(* PLC project Export.project, CODESYS CODESYS V3.5 SP19 Patch 7 *)
(* stored: creationDateTime 2025-04-03T07:54:30.183, modificationDateTime 2025-04-03T07:54:30.183 *)

VAR_GLOBAL  (* GVL_ClimateControl *)
  typClimateControllerInterfaceRoom401 : typMultiModeClimateControl_00_01;
  typClimateControllerInterfaceRoom406 : typMultiModeClimateControl_00_01;
  typClimateControllerInterfaceRoom407 : typMultiModeClimateControl_00_01;
  typClimateControllerInterfaceRoom408 : typMultiModeClimateControl_00_01;
  typClimateControllerInterfaceRoom409 : typMultiModeClimateControl_00_01;
  typClimateControllerInterfaceRoom464 : typMultiModeClimateControl_00_01;
  typClimateControllerInterfaceRoom415 : typMultiModeClimateControl_00_01;
  typClimateControllerInterfaceRoom422 : typMultiModeClimateControl_00_01;
  typClimateControllerInterfaceRoom426_1 : typMultiModeClimateControl_00_01;
  typClimateControllerInterfaceRoom426_2 : typMultiModeClimateControl_00_01;
  typClimateControllerInterfaceRoom426_3 : typMultiModeClimateControl_00_01;
  typClimateControllerInterfaceRoom528 : typMultiModeClimateControl_00_01;
  typClimateControllerInterfaceRoom523 : typMultiModeClimateControl_00_01;
  typClimateControllerInterfaceRoom531 : typMultiModeClimateControl_00_01;
  typClimateControllerInterfaceRoom535_1 : typMultiModeClimateControl_00_01;
  typClimateControllerInterfaceRoom535_2 : typMultiModeClimateControl_00_01;
  typClimateControllerInterfaceRoom535_3 : typMultiModeClimateControl_00_01;
  typClimateControllerInterfaceRoom536 : typMultiModeClimateControl_00_01;
  typClimateControllerInterfaceRoom543 : typMultiModeClimateControl_00_01;
  typClimateControllerInterfaceRoom547_1 : typMultiModeClimateControl_00_01;
  typClimateControllerInterfaceRoom547_2 : typMultiModeClimateControl_00_01;
  typClimateControllerInterfaceRoom544 : typMultiModeClimateControl_00_01;
  SLETT_MEG : BOOL;  (* Kopier til PersistentVars! *)
  typClimateControllerSettingsRoom401 : typMultiModeClimateControlSettings_00_01;
  typClimateControllerSettingsRoom406 : typMultiModeClimateControlSettings_00_01;
  typClimateControllerSettingsRoom407 : typMultiModeClimateControlSettings_00_01;
  typClimateControllerSettingsRoom408 : typMultiModeClimateControlSettings_00_01;
  typClimateControllerSettingsRoom409 : typMultiModeClimateControlSettings_00_01;
  typClimateControllerSettingsRoom464 : typMultiModeClimateControlSettings_00_01;
  typClimateControllerSettingsRoom415 : typMultiModeClimateControlSettings_00_01;
  typClimateControllerSettingsRoom422 : typMultiModeClimateControlSettings_00_01;
  typClimateControllerSettingsRoom426_1 : typMultiModeClimateControlSettings_00_01;
  typClimateControllerSettingsRoom426_2 : typMultiModeClimateControlSettings_00_01;
  typClimateControllerSettingsRoom426_3 : typMultiModeClimateControlSettings_00_01;
  typClimateControllerSettingsRoom528 : typMultiModeClimateControlSettings_00_01;
  typClimateControllerSettingsRoom523 : typMultiModeClimateControlSettings_00_01;
  typClimateControllerSettingsRoom531 : typMultiModeClimateControlSettings_00_01;
  typClimateControllerSettingsRoom535_1 : typMultiModeClimateControlSettings_00_01;
  typClimateControllerSettingsRoom535_2 : typMultiModeClimateControlSettings_00_01;
  typClimateControllerSettingsRoom535_3 : typMultiModeClimateControlSettings_00_01;
  typClimateControllerSettingsRoom536 : typMultiModeClimateControlSettings_00_01;
  typClimateControllerSettingsRoom543 : typMultiModeClimateControlSettings_00_01;
  typClimateControllerSettingsRoom547_1 : typMultiModeClimateControlSettings_00_01;
  typClimateControllerSettingsRoom547_2 : typMultiModeClimateControlSettings_00_01;
  typClimateControllerSettingsRoom544 : typMultiModeClimateControlSettings_00_01;
END_VAR

VAR_GLOBAL  (* GVL_BACnet *)
  C_5640_501_06_RBA01_D_R0401 : FbBinaryOutput_Medium (0) := (                _sDescription := 'Tilstedeværelsesdetektor',                 _sActiveText := 'Tilstedeværelse',                 _sInactiveText := 'Ingen tilstedeværelse'           );
  C_5640_501_06_RTC01_MV_R0401 : FbAnalogInput_Large (0) := (                _sDescription := 'Målt temperatur',                 _rCov_Increment := 0.1,                 _eUnits := WagoTypesBacnet.eBACnetUnits.UNIT_DEGREES_C,                 _rHighLimit := 28,                 _ILimitEnable := ( xLowLimitReporting := FALSE, xHighLimitReporting := TRUE ),                 _udiNotificationClass := 22           );
  C_5640_501_06_RTC01_SPV_R0401 : FbAnalogValue_Medium (0) := (                _sDescription := 'Arbeidende settpunkt',                 _rCov_Increment := 0.1,                 _eUnits := WagoTypesBacnet.eBACnetUnits.UNIT_DEGREES_C           );
  C_5640_501_06_RTC01_SPV_Komf_R0401 : FbAnalogValue_Medium (1) := (                _sDescription := 'Settpunkt komfort',                 _rCov_Increment := 0.1,                 _eUnits := WagoTypesBacnet.eBACnetUnits.UNIT_DEGREES_C           );
  C_5640_501_06_RTC01_SPV_Stdb_R0401 : FbAnalogValue_Medium (2) := (                _sDescription := 'Settpunkt Standby',                 _rCov_Increment := 0.1,                 _eUnits := WagoTypesBacnet.eBACnetUnits.UNIT_DEGREES_C           );
  C_5640_501_06_RTC01_SPV_Natt_R0401 : FbAnalogValue_Medium (3) := (                _sDescription := 'Settpunkt Natt',                 _rCov_Increment := 0.1,                 _eUnits := WagoTypesBacnet.eBACnetUnits.UNIT_DEGREES_C           );
  C_5640_501_06_RTC01_MOD_FB_R0401 : FbMultiStateValue_Large (0) := (                _sDescription := 'Tilbakemelding driftmodus',                 _udiNumberOfStates := 5,                 _xEventDetectionEnable := FALSE,                 _udiNotificationClass := 99           );
  C_5640_501_06_RTC01_KMD_MSV_R0401 : FbMultiStateValue_Large (1) := (                _sDescription := 'Kalender',                 _udiNumberOfStates := 10,                 _xEventDetectionEnable := FALSE,                 _udiNotificationClass := 99           );
  C_5640_501_06_RTC01_SP_Tid_Stdb_R0401 : FbAnalogValue_Medium (4) := (                _sDescription := 'Utløpstid tilstedeværelse',                 _rCov_Increment := 1,                 _eUnits := WagoTypesBacnet.eBACnetUnits.UNIT_MINUTES           );
  C_5640_501_06_RYA601_SP_R0401 : FbAnalogValue_Medium (5) := (                _sDescription := 'Settpunkt',                 _rCov_Increment := 1,                 _eUnits := WagoTypesBacnet.eBACnetUnits.UNIT_PARTS_PER_MILLION           );
  C_5640_501_06_RYA601_MV_R0401 : FbAnalogInput_Large (1) := (                _sDescription := 'Målt CO2-konsentrasjon',                 _rCov_Increment := 1,                 _eUnits := WagoTypesBacnet.eBACnetUnits.UNIT_PARTS_PER_MILLION,                 _rHighLimit := 1000,                 _ILimitEnable := ( xLowLimitReporting := FALSE, xHighLimitReporting := TRUE ),                 _udiNotificationClass := 22           );
  C_5640_501_06_SBB01_C_R0401 : FbAnalogOutput_Medium (0) := (                _sDescription := 'Pådrag varmeorgan',                 _rCov_Increment := 1,                 _eUnits := WagoTypesBacnet.eBACnetUnits.UNIT_PERCENT           );
  C_5640_501_06_RBA01_D_R0406 : FbBinaryOutput_Medium (1) := (                _sDescription := 'Tilstedeværelsesdetektor',                 _sActiveText := 'Tilstedeværelse',                 _sInactiveText := 'Ingen tilstedeværelse'           );
  C_5640_501_06_RTC01_MV_R0406 : FbAnalogInput_Large (2) := (                _sDescription := 'Målt temperatur',                 _rCov_Increment := 0.1,                 _eUnits := WagoTypesBacnet.eBACnetUnits.UNIT_DEGREES_C,                 _rHighLimit := 28,                 _ILimitEnable := ( xLowLimitReporting := FALSE, xHighLimitReporting := TRUE ),                 _udiNotificationClass := 22           );
  C_5640_501_06_RTC01_SPV_R0406 : FbAnalogValue_Medium (6) := (                _sDescription := 'Arbeidende settpunkt',                 _rCov_Increment := 0.1,                 _eUnits := WagoTypesBacnet.eBACnetUnits.UNIT_DEGREES_C           );
  C_5640_501_06_RTC01_SPV_Komf_R0406 : FbAnalogValue_Medium (7) := (                _sDescription := 'Settpunkt komfort',                 _rCov_Increment := 0.1,                 _eUnits := WagoTypesBacnet.eBACnetUnits.UNIT_DEGREES_C           );
  C_5640_501_06_RTC01_SPV_Stdb_R0406 : FbAnalogValue_Medium (8) := (                _sDescription := 'Settpunkt Standby',                 _rCov_Increment := 0.1,                 _eUnits := WagoTypesBacnet.eBACnetUnits.UNIT_DEGREES_C           );
  C_5640_501_06_RTC01_SPV_Natt_R0406 : FbAnalogValue_Medium (9) := (                _sDescription := 'Settpunkt Natt',                 _rCov_Increment := 0.1,                 _eUnits := WagoTypesBacnet.eBACnetUnits.UNIT_DEGREES_C           );
  C_5640_501_06_RTC01_MOD_FB_R0406 : FbMultiStateValue_Large (2) := (                _sDescription := 'Tilbakemelding driftmodus',                 _udiNumberOfStates := 5,                 _xEventDetectionEnable := FALSE,                 _udiNotificationClass := 99           );
  C_5640_501_06_RTC01_KMD_MSV_R0406 : FbMultiStateValue_Large (3) := (                _sDescription := 'Kalender',                 _udiNumberOfStates := 10,                 _xEventDetectionEnable := FALSE,                 _udiNotificationClass := 99           );
  C_5640_501_06_RTC01_SP_Tid_Stdb_R0406 : FbAnalogValue_Medium (10) := (                _sDescription := 'Utløpstid tilstedeværelse',                 _rCov_Increment := 1,                 _eUnits := WagoTypesBacnet.eBACnetUnits.UNIT_MINUTES           );
  C_5640_501_06_RYA601_SP_R0406 : FbAnalogValue_Medium (11) := (                _sDescription := 'Settpunkt',                 _rCov_Increment := 1,                 _eUnits := WagoTypesBacnet.eBACnetUnits.UNIT_PARTS_PER_MILLION           );
  C_5640_501_06_RYA601_MV_R0406 : FbAnalogInput_Large (3) := (                _sDescription := 'Målt CO2-konsentrasjon',                 _rCov_Increment := 1,                 _eUnits := WagoTypesBacnet.eBACnetUnits.UNIT_PARTS_PER_MILLION,                 _rHighLimit := 1000,                 _ILimitEnable := ( xLowLimitReporting := FALSE, xHighLimitReporting := TRUE ),                 _udiNotificationClass := 22           );
  C_5640_501_06_SBB01_C_R0406 : FbAnalogOutput_Medium (1) := (                _sDescription := 'Pådrag varmeorgan',                 _rCov_Increment := 1,                 _eUnits := WagoTypesBacnet.eBACnetUnits.UNIT_PERCENT           );
  C_5640_501_06_RBA01_D_R0407 : FbBinaryOutput_Medium (2) := (                _sDescription := 'Tilstedeværelsesdetektor',                 _sActiveText := 'Tilstedeværelse',                 _sInactiveText := 'Ingen tilstedeværelse'           );
  C_5640_501_06_RTC01_MV_R0407 : FbAnalogInput_Large (4) := (                _sDescription := 'Målt temperatur',                 _rCov_Increment := 0.1,                 _eUnits := WagoTypesBacnet.eBACnetUnits.UNIT_DEGREES_C,                 _rHighLimit := 28,                 _ILimitEnable := ( xLowLimitReporting := FALSE, xHighLimitReporting := TRUE ),                 _udiNotificationClass := 22           );
  C_5640_501_06_RTC01_SPV_R0407 : FbAnalogValue_Medium (12) := (                _sDescription := 'Arbeidende settpunkt',                 _rCov_Increment := 0.1,                 _eUnits := WagoTypesBacnet.eBACnetUnits.UNIT_DEGREES_C           );
  C_5640_501_06_RTC01_SPV_Komf_R0407 : FbAnalogValue_Medium (13) := (                _sDescription := 'Settpunkt komfort',                 _rCov_Increment := 0.1,                 _eUnits := WagoTypesBacnet.eBACnetUnits.UNIT_DEGREES_C           );
  C_5640_501_06_RTC01_SPV_Stdb_R0407 : FbAnalogValue_Medium (14) := (                _sDescription := 'Settpunkt Standby',                 _rCov_Increment := 0.1,                 _eUnits := WagoTypesBacnet.eBACnetUnits.UNIT_DEGREES_C           );
  C_5640_501_06_RTC01_SPV_Natt_R0407 : FbAnalogValue_Medium (15) := (                _sDescription := 'Settpunkt Natt',                 _rCov_Increment := 0.1,                 _eUnits := WagoTypesBacnet.eBACnetUnits.UNIT_DEGREES_C           );
  C_5640_501_06_RTC01_MOD_FB_R0407 : FbMultiStateValue_Large (4) := (                _sDescription := 'Tilbakemelding driftmodus',                 _udiNumberOfStates := 5,                 _xEventDetectionEnable := FALSE,                 _udiNotificationClass := 99           );
  C_5640_501_06_RTC01_KMD_MSV_R0407 : FbMultiStateValue_Large (5) := (                _sDescription := 'Kalender',                 _udiNumberOfStates := 10,                 _xEventDetectionEnable := FALSE,                 _udiNotificationClass := 99           );
  C_5640_501_06_RTC01_SP_Tid_Stdb_R0407 : FbAnalogValue_Medium (16) := (                _sDescription := 'Utløpstid tilstedeværelse',                 _rCov_Increment := 1,                 _eUnits := WagoTypesBacnet.eBACnetUnits.UNIT_MINUTES           );
  C_5640_501_06_RYA601_SP_R0407 : FbAnalogValue_Medium (17) := (                _sDescription := 'Settpunkt',                 _rCov_Increment := 1,                 _eUnits := WagoTypesBacnet.eBACnetUnits.UNIT_PARTS_PER_MILLION           );
  C_5640_501_06_RYA601_MV_R0407 : FbAnalogInput_Large (5) := (                _sDescription := 'Målt CO2-konsentrasjon',                 _rCov_Increment := 1,                 _eUnits := WagoTypesBacnet.eBACnetUnits.UNIT_PARTS_PER_MILLION,                 _rHighLimit := 1000,                 _ILimitEnable := ( xLowLimitReporting := FALSE, xHighLimitReporting := TRUE ),                 _udiNotificationClass := 22           );
  C_5640_501_06_SBB01_C_R0407 : FbAnalogOutput_Medium (2) := (                _sDescription := 'Pådrag varmeorgan',                 _rCov_Increment := 1,                 _eUnits := WagoTypesBacnet.eBACnetUnits.UNIT_PERCENT           );
  C_5640_501_06_RBA01_D_R0408 : FbBinaryOutput_Medium (3) := (                _sDescription := 'Tilstedeværelsesdetektor',                 _sActiveText := 'Tilstedeværelse',                 _sInactiveText := 'Ingen tilstedeværelse'           );
  C_5640_501_06_RTC01_MV_R0408 : FbAnalogInput_Large (6) := (                _sDescription := 'Målt temperatur',                 _rCov_Increment := 0.1,                 _eUnits := WagoTypesBacnet.eBACnetUnits.UNIT_DEGREES_C,                 _rHighLimit := 28,                 _ILimitEnable := ( xLowLimitReporting := FALSE, xHighLimitReporting := TRUE ),                 _udiNotificationClass := 22           );
  C_5640_501_06_RTC01_SPV_R0408 : FbAnalogValue_Medium (18) := (                _sDescription := 'Arbeidende settpunkt',                 _rCov_Increment := 0.1,                 _eUnits := WagoTypesBacnet.eBACnetUnits.UNIT_DEGREES_C           );
  C_5640_501_06_RTC01_SPV_Komf_R0408 : FbAnalogValue_Medium (19) := (                _sDescription := 'Settpunkt komfort',                 _rCov_Increment := 0.1,                 _eUnits := WagoTypesBacnet.eBACnetUnits.UNIT_DEGREES_C           );
  C_5640_501_06_RTC01_SPV_Stdb_R0408 : FbAnalogValue_Medium (20) := (                _sDescription := 'Settpunkt Standby',                 _rCov_Increment := 0.1,                 _eUnits := WagoTypesBacnet.eBACnetUnits.UNIT_DEGREES_C           );
  C_5640_501_06_RTC01_SPV_Natt_R0408 : FbAnalogValue_Medium (21) := (                _sDescription := 'Settpunkt Natt',                 _rCov_Increment := 0.1,                 _eUnits := WagoTypesBacnet.eBACnetUnits.UNIT_DEGREES_C           );
  C_5640_501_06_RTC01_MOD_FB_R0408 : FbMultiStateValue_Large (6) := (                _sDescription := 'Tilbakemelding driftmodus',                 _udiNumberOfStates := 5,                 _xEventDetectionEnable := FALSE,                 _udiNotificationClass := 99           );
  C_5640_501_06_RTC01_KMD_MSV_R0408 : FbMultiStateValue_Large (7) := (                _sDescription := 'Kalender',                 _udiNumberOfStates := 10,                 _xEventDetectionEnable := FALSE,                 _udiNotificationClass := 99           );
  C_5640_501_06_RTC01_SP_Tid_Stdb_R0408 : FbAnalogValue_Medium (22) := (                _sDescription := 'Utløpstid tilstedeværelse',                 _rCov_Increment := 1,                 _eUnits := WagoTypesBacnet.eBACnetUnits.UNIT_MINUTES           );
  C_5640_501_06_RYA601_SP_R0408 : FbAnalogValue_Medium (23) := (                _sDescription := 'Settpunkt',                 _rCov_Increment := 1,                 _eUnits := WagoTypesBacnet.eBACnetUnits.UNIT_PARTS_PER_MILLION           );
  C_5640_501_06_RYA601_MV_R0408 : FbAnalogInput_Large (7) := (                _sDescription := 'Målt CO2-konsentrasjon',                 _rCov_Increment := 1,                 _eUnits := WagoTypesBacnet.eBACnetUnits.UNIT_PARTS_PER_MILLION,                 _rHighLimit := 1000,                 _ILimitEnable := ( xLowLimitReporting := FALSE, xHighLimitReporting := TRUE ),                 _udiNotificationClass := 22           );
  C_5640_501_06_SBB01_C_R0408 : FbAnalogOutput_Medium (3) := (                _sDescription := 'Pådrag varmeorgan',                 _rCov_Increment := 1,                 _eUnits := WagoTypesBacnet.eBACnetUnits.UNIT_PERCENT           );
  C_5640_501_06_RBA01_D_R0409 : FbBinaryOutput_Medium (4) := (                _sDescription := 'Tilstedeværelsesdetektor',                 _sActiveText := 'Tilstedeværelse',                 _sInactiveText := 'Ingen tilstedeværelse'           );
  C_5640_501_06_RTC01_MV_R0409 : FbAnalogInput_Large (8) := (                _sDescription := 'Målt temperatur',                 _rCov_Increment := 0.1,                 _eUnits := WagoTypesBacnet.eBACnetUnits.UNIT_DEGREES_C,                 _rHighLimit := 28,                 _ILimitEnable := ( xLowLimitReporting := FALSE, xHighLimitReporting := TRUE ),                 _udiNotificationClass := 22           );
  C_5640_501_06_RTC01_SPV_R0409 : FbAnalogValue_Medium (24) := (                _sDescription := 'Arbeidende settpunkt',                 _rCov_Increment := 0.1,                 _eUnits := WagoTypesBacnet.eBACnetUnits.UNIT_DEGREES_C           );
  C_5640_501_06_RTC01_SPV_Komf_R0409 : FbAnalogValue_Medium (25) := (                _sDescription := 'Settpunkt komfort',                 _rCov_Increment := 0.1,                 _eUnits := WagoTypesBacnet.eBACnetUnits.UNIT_DEGREES_C           );
  C_5640_501_06_RTC01_SPV_Stdb_R0409 : FbAnalogValue_Medium (26) := (                _sDescription := 'Settpunkt Standby',                 _rCov_Increment := 0.1,                 _eUnits := WagoTypesBacnet.eBACnetUnits.UNIT_DEGREES_C           );
  C_5640_501_06_RTC01_SPV_Natt_R0409 : FbAnalogValue_Medium (27) := (                _sDescription := 'Settpunkt Natt',                 _rCov_Increment := 0.1,                 _eUnits := WagoTypesBacnet.eBACnetUnits.UNIT_DEGREES_C           );
  C_5640_501_06_RTC01_MOD_FB_R0409 : FbMultiStateValue_Large (8) := (                _sDescription := 'Tilbakemelding driftmodus',                 _udiNumberOfStates := 5,                 _xEventDetectionEnable := FALSE,                 _udiNotificationClass := 99           );
  C_5640_501_06_RTC01_KMD_MSV_R0409 : FbMultiStateValue_Large (9) := (                _sDescription := 'Kalender',                 _udiNumberOfStates := 10,                 _xEventDetectionEnable := FALSE,                 _udiNotificationClass := 99           );
  C_5640_501_06_RTC01_SP_Tid_Stdb_R0409 : FbAnalogValue_Medium (28) := (                _sDescription := 'Utløpstid tilstedeværelse',                 _rCov_Increment := 1,                 _eUnits := WagoTypesBacnet.eBACnetUnits.UNIT_MINUTES           );
  C_5640_501_06_RYA601_SP_R0409 : FbAnalogValue_Medium (29) := (                _sDescription := 'Settpunkt',                 _rCov_Increment := 1,                 _eUnits := WagoTypesBacnet.eBACnetUnits.UNIT_PARTS_PER_MILLION           );
  C_5640_501_06_RYA601_MV_R0409 : FbAnalogInput_Large (9) := (                _sDescription := 'Målt CO2-konsentrasjon',                 _rCov_Increment := 1,                 _eUnits := WagoTypesBacnet.eBACnetUnits.UNIT_PARTS_PER_MILLION,                 _rHighLimit := 1000,                 _ILimitEnable := ( xLowLimitReporting := FALSE, xHighLimitReporting := TRUE ),                 _udiNotificationClass := 22           );
  C_5640_501_06_SBB01_C_R0409 : FbAnalogOutput_Medium (4) := (                _sDescription := 'Pådrag varmeorgan',                 _rCov_Increment := 1,                 _eUnits := WagoTypesBacnet.eBACnetUnits.UNIT_PERCENT           );
  C_5640_501_06_RBA01_D_R0464 : FbBinaryOutput_Medium (5) := (                _sDescription := 'Tilstedeværelsesdetektor',                 _sActiveText := 'Tilstedeværelse',                 _sInactiveText := 'Ingen tilstedeværelse'           );
  C_5640_501_06_RTC01_MV_R0464 : FbAnalogInput_Large (10) := (                _sDescription := 'Målt temperatur',                 _rCov_Increment := 0.1,                 _eUnits := WagoTypesBacnet.eBACnetUnits.UNIT_DEGREES_C,                 _rHighLimit := 28,                 _ILimitEnable := ( xLowLimitReporting := FALSE, xHighLimitReporting := TRUE ),                 _udiNotificationClass := 22           );
  C_5640_501_06_RTC01_SPV_R0464 : FbAnalogValue_Medium (30) := (                _sDescription := 'Arbeidende settpunkt',                 _rCov_Increment := 0.1,                 _eUnits := WagoTypesBacnet.eBACnetUnits.UNIT_DEGREES_C           );
  C_5640_501_06_RTC01_SPV_Komf_R0464 : FbAnalogValue_Medium (31) := (                _sDescription := 'Settpunkt komfort',                 _rCov_Increment := 0.1,                 _eUnits := WagoTypesBacnet.eBACnetUnits.UNIT_DEGREES_C           );
  C_5640_501_06_RTC01_SPV_Stdb_R0464 : FbAnalogValue_Medium (32) := (                _sDescription := 'Settpunkt Standby',                 _rCov_Increment := 0.1,                 _eUnits := WagoTypesBacnet.eBACnetUnits.UNIT_DEGREES_C           );
  C_5640_501_06_RTC01_SPV_Natt_R0464 : FbAnalogValue_Medium (33) := (                _sDescription := 'Settpunkt Natt',                 _rCov_Increment := 0.1,                 _eUnits := WagoTypesBacnet.eBACnetUnits.UNIT_DEGREES_C           );
  C_5640_501_06_RTC01_MOD_FB_R0464 : FbMultiStateValue_Large (10) := (                _sDescription := 'Tilbakemelding driftmodus',                 _udiNumberOfStates := 5,                 _xEventDetectionEnable := FALSE,                 _udiNotificationClass := 99           );
  C_5640_501_06_RTC01_KMD_MSV_R0464 : FbMultiStateValue_Large (11) := (                _sDescription := 'Kalender',                 _udiNumberOfStates := 10,                 _xEventDetectionEnable := FALSE,                 _udiNotificationClass := 99           );
  C_5640_501_06_RTC01_SP_Tid_Stdb_R0464 : FbAnalogValue_Medium (34) := (                _sDescription := 'Utløpstid tilstedeværelse',                 _rCov_Increment := 1,                 _eUnits := WagoTypesBacnet.eBACnetUnits.UNIT_MINUTES           );
  C_5640_501_06_RYA601_SP_R0464 : FbAnalogValue_Medium (35) := (                _sDescription := 'Settpunkt',                 _rCov_Increment := 1,                 _eUnits := WagoTypesBacnet.eBACnetUnits.UNIT_PARTS_PER_MILLION           );
  C_5640_501_06_RYA601_MV_R0464 : FbAnalogInput_Large (11) := (                _sDescription := 'Målt CO2-konsentrasjon',                 _rCov_Increment := 1,                 _eUnits := WagoTypesBacnet.eBACnetUnits.UNIT_PARTS_PER_MILLION,                 _rHighLimit := 1000,                 _ILimitEnable := ( xLowLimitReporting := FALSE, xHighLimitReporting := TRUE ),                 _udiNotificationClass := 22           );
  C_5640_501_06_SBB01_C_R0464 : FbAnalogOutput_Medium (5) := (                _sDescription := 'Pådrag varmeorgan',                 _rCov_Increment := 1,                 _eUnits := WagoTypesBacnet.eBACnetUnits.UNIT_PERCENT           );
  C_5640_501_06_RBA01_D_R0415 : FbBinaryOutput_Medium (6) := (                _sDescription := 'Tilstedeværelsesdetektor',                 _sActiveText := 'Tilstedeværelse',                 _sInactiveText := 'Ingen tilstedeværelse'           );
  C_5640_501_06_RTC01_MV_R0415 : FbAnalogInput_Large (12) := (                _sDescription := 'Målt temperatur',                 _rCov_Increment := 0.1,                 _eUnits := WagoTypesBacnet.eBACnetUnits.UNIT_DEGREES_C,                 _rHighLimit := 28,                 _ILimitEnable := ( xLowLimitReporting := FALSE, xHighLimitReporting := TRUE ),                 _udiNotificationClass := 22           );
  C_5640_501_06_RTC01_SPV_R0415 : FbAnalogValue_Medium (36) := (                _sDescription := 'Arbeidende settpunkt',                 _rCov_Increment := 0.1,                 _eUnits := WagoTypesBacnet.eBACnetUnits.UNIT_DEGREES_C           );
  C_5640_501_06_RTC01_SPV_Komf_R0415 : FbAnalogValue_Medium (37) := (                _sDescription := 'Settpunkt komfort',                 _rCov_Increment := 0.1,                 _eUnits := WagoTypesBacnet.eBACnetUnits.UNIT_DEGREES_C           );
  C_5640_501_06_RTC01_SPV_Stdb_R0415 : FbAnalogValue_Medium (38) := (                _sDescription := 'Settpunkt Standby',                 _rCov_Increment := 0.1,                 _eUnits := WagoTypesBacnet.eBACnetUnits.UNIT_DEGREES_C           );
  C_5640_501_06_RTC01_SPV_Natt_R0415 : FbAnalogValue_Medium (39) := (                _sDescription := 'Settpunkt Natt',                 _rCov_Increment := 0.1,                 _eUnits := WagoTypesBacnet.eBACnetUnits.UNIT_DEGREES_C           );
  C_5640_501_06_RTC01_MOD_FB_R0415 : FbMultiStateValue_Large (12) := (                _sDescription := 'Tilbakemelding driftmodus',                 _udiNumberOfStates := 5,                 _xEventDetectionEnable := FALSE,                 _udiNotificationClass := 99           );
  C_5640_501_06_RTC01_KMD_MSV_R0415 : FbMultiStateValue_Large (13) := (                _sDescription := 'Kalender',                 _udiNumberOfStates := 10,                 _xEventDetectionEnable := FALSE,                 _udiNotificationClass := 99           );
  C_5640_501_06_RTC01_SP_Tid_Stdb_R0415 : FbAnalogValue_Medium (40) := (                _sDescription := 'Utløpstid tilstedeværelse',                 _rCov_Increment := 1,                 _eUnits := WagoTypesBacnet.eBACnetUnits.UNIT_MINUTES           );
  C_5640_501_06_RYA601_SP_R0415 : FbAnalogValue_Medium (41) := (                _sDescription := 'Settpunkt',                 _rCov_Increment := 1,                 _eUnits := WagoTypesBacnet.eBACnetUnits.UNIT_PARTS_PER_MILLION           );
  C_5640_501_06_RYA601_MV_R0415 : FbAnalogInput_Large (13) := (                _sDescription := 'Målt CO2-konsentrasjon',                 _rCov_Increment := 1,                 _eUnits := WagoTypesBacnet.eBACnetUnits.UNIT_PARTS_PER_MILLION,                 _rHighLimit := 1000,                 _ILimitEnable := ( xLowLimitReporting := FALSE, xHighLimitReporting := TRUE ),                 _udiNotificationClass := 22           );
  C_5640_501_06_SBB01_C_R0415 : FbAnalogOutput_Medium (6) := (                _sDescription := 'Pådrag varmeorgan',                 _rCov_Increment := 1,                 _eUnits := WagoTypesBacnet.eBACnetUnits.UNIT_PERCENT           );
  C_5640_501_06_RBA01_D_R0422 : FbBinaryOutput_Medium (7) := (                _sDescription := 'Tilstedeværelsesdetektor',                 _sActiveText := 'Tilstedeværelse',                 _sInactiveText := 'Ingen tilstedeværelse'           );
  C_5640_501_06_RTC01_MV_R0422 : FbAnalogInput_Large (14) := (                _sDescription := 'Målt temperatur',                 _rCov_Increment := 0.1,                 _eUnits := WagoTypesBacnet.eBACnetUnits.UNIT_DEGREES_C,                 _rHighLimit := 28,                 _ILimitEnable := ( xLowLimitReporting := FALSE, xHighLimitReporting := TRUE ),                 _udiNotificationClass := 22           );
  C_5640_501_06_RTC01_SPV_R0422 : FbAnalogValue_Medium (42) := (                _sDescription := 'Arbeidende settpunkt',                 _rCov_Increment := 0.1,                 _eUnits := WagoTypesBacnet.eBACnetUnits.UNIT_DEGREES_C           );
  C_5640_501_06_RTC01_SPV_Komf_R0422 : FbAnalogValue_Medium (43) := (                _sDescription := 'Settpunkt komfort',                 _rCov_Increment := 0.1,                 _eUnits := WagoTypesBacnet.eBACnetUnits.UNIT_DEGREES_C           );
  C_5640_501_06_RTC01_SPV_Stdb_R0422 : FbAnalogValue_Medium (44) := (                _sDescription := 'Settpunkt Standby',                 _rCov_Increment := 0.1,                 _eUnits := WagoTypesBacnet.eBACnetUnits.UNIT_DEGREES_C           );
  C_5640_501_06_RTC01_SPV_Natt_R0422 : FbAnalogValue_Medium (45) := (                _sDescription := 'Settpunkt Natt',                 _rCov_Increment := 0.1,                 _eUnits := WagoTypesBacnet.eBACnetUnits.UNIT_DEGREES_C           );
  C_5640_501_06_RTC01_MOD_FB_R0422 : FbMultiStateValue_Large (14) := (                _sDescription := 'Tilbakemelding driftmodus',                 _udiNumberOfStates := 5,                 _xEventDetectionEnable := FALSE,                 _udiNotificationClass := 99           );
  C_5640_501_06_RTC01_KMD_MSV_R0422 : FbMultiStateValue_Large (15) := (                _sDescription := 'Kalender',                 _udiNumberOfStates := 10,                 _xEventDetectionEnable := FALSE,                 _udiNotificationClass := 99           );
  C_5640_501_06_RTC01_SP_Tid_Stdb_R0422 : FbAnalogValue_Medium (46) := (                _sDescription := 'Utløpstid tilstedeværelse',                 _rCov_Increment := 1,                 _eUnits := WagoTypesBacnet.eBACnetUnits.UNIT_MINUTES           );
  C_5640_501_06_RYA601_SP_R0422 : FbAnalogValue_Medium (47) := (                _sDescription := 'Settpunkt',                 _rCov_Increment := 1,                 _eUnits := WagoTypesBacnet.eBACnetUnits.UNIT_PARTS_PER_MILLION           );
  C_5640_501_06_RYA601_MV_R0422 : FbAnalogInput_Large (15) := (                _sDescription := 'Målt CO2-konsentrasjon',                 _rCov_Increment := 1,                 _eUnits := WagoTypesBacnet.eBACnetUnits.UNIT_PARTS_PER_MILLION,                 _rHighLimit := 1000,                 _ILimitEnable := ( xLowLimitReporting := FALSE, xHighLimitReporting := TRUE ),                 _udiNotificationClass := 22           );
  C_5640_501_06_SBB01_C_R0422 : FbAnalogOutput_Medium (7) := (                _sDescription := 'Pådrag varmeorgan',                 _rCov_Increment := 1,                 _eUnits := WagoTypesBacnet.eBACnetUnits.UNIT_PERCENT           );
  C_5640_501_06_RBA01_D_R0426_1 : FbBinaryOutput_Medium (8) := (                _sDescription := 'Tilstedeværelsesdetektor',                 _sActiveText := 'Tilstedeværelse',                 _sInactiveText := 'Ingen tilstedeværelse'           );
  C_5640_501_06_RTC01_MV_R0426_1 : FbAnalogInput_Large (16) := (                _sDescription := 'Målt temperatur',                 _rCov_Increment := 0.1,                 _eUnits := WagoTypesBacnet.eBACnetUnits.UNIT_DEGREES_C,                 _rHighLimit := 28,                 _ILimitEnable := ( xLowLimitReporting := FALSE, xHighLimitReporting := TRUE ),                 _udiNotificationClass := 22           );
  C_5640_501_06_RTC01_SPV_R0426_1 : FbAnalogValue_Medium (48) := (                _sDescription := 'Arbeidende settpunkt',                 _rCov_Increment := 0.1,                 _eUnits := WagoTypesBacnet.eBACnetUnits.UNIT_DEGREES_C           );
  C_5640_501_06_RTC01_SPV_Komf_R0426_1 : FbAnalogValue_Medium (49) := (                _sDescription := 'Settpunkt komfort',                 _rCov_Increment := 0.1,                 _eUnits := WagoTypesBacnet.eBACnetUnits.UNIT_DEGREES_C           );
  C_5640_501_06_RTC01_SPV_Stdb_R0426_1 : FbAnalogValue_Medium (50) := (                _sDescription := 'Settpunkt Standby',                 _rCov_Increment := 0.1,                 _eUnits := WagoTypesBacnet.eBACnetUnits.UNIT_DEGREES_C           );
  C_5640_501_06_RTC01_SPV_Natt_R0426_1 : FbAnalogValue_Medium (51) := (                _sDescription := 'Settpunkt Natt',                 _rCov_Increment := 0.1,                 _eUnits := WagoTypesBacnet.eBACnetUnits.UNIT_DEGREES_C           );
  C_5640_501_06_RTC01_MOD_FB_R0426_1 : FbMultiStateValue_Large (16) := (                _sDescription := 'Tilbakemelding driftmodus',                 _udiNumberOfStates := 5,                 _xEventDetectionEnable := FALSE,                 _udiNotificationClass := 99           );
  C_5640_501_06_RTC01_KMD_MSV_R0426_1 : FbMultiStateValue_Large (17) := (                _sDescription := 'Kalender',                 _udiNumberOfStates := 10,                 _xEventDetectionEnable := FALSE,                 _udiNotificationClass := 99           );
  C_5640_501_06_RTC01_SP_Tid_Stdb_R0426_1 : FbAnalogValue_Medium (52) := (                _sDescription := 'Utløpstid tilstedeværelse',                 _rCov_Increment := 1,                 _eUnits := WagoTypesBacnet.eBACnetUnits.UNIT_MINUTES           );
  C_5640_501_06_RYA601_SP_R0426_1 : FbAnalogValue_Medium (53) := (                _sDescription := 'Settpunkt',                 _rCov_Increment := 1,                 _eUnits := WagoTypesBacnet.eBACnetUnits.UNIT_PARTS_PER_MILLION           );
  C_5640_501_06_RYA601_MV_R0426_1 : FbAnalogInput_Large (17) := (                _sDescription := 'Målt CO2-konsentrasjon',                 _rCov_Increment := 1,                 _eUnits := WagoTypesBacnet.eBACnetUnits.UNIT_PARTS_PER_MILLION,                 _rHighLimit := 1000,                 _ILimitEnable := ( xLowLimitReporting := FALSE, xHighLimitReporting := TRUE ),                 _udiNotificationClass := 22           );
  C_5640_501_06_SBB01_C_R0426_1 : FbAnalogOutput_Medium (8) := (                _sDescription := 'Pådrag varmeorgan',                 _rCov_Increment := 1,                 _eUnits := WagoTypesBacnet.eBACnetUnits.UNIT_PERCENT           );
  C_5640_501_06_RBA01_D_R0426_2 : FbBinaryOutput_Medium (9) := (                _sDescription := 'Tilstedeværelsesdetektor',                 _sActiveText := 'Tilstedeværelse',                 _sInactiveText := 'Ingen tilstedeværelse'           );
  C_5640_501_06_RTC01_MV_R0426_2 : FbAnalogInput_Large (18) := (                _sDescription := 'Målt temperatur',                 _rCov_Increment := 0.1,                 _eUnits := WagoTypesBacnet.eBACnetUnits.UNIT_DEGREES_C,                 _rHighLimit := 28,                 _ILimitEnable := ( xLowLimitReporting := FALSE, xHighLimitReporting := TRUE ),                 _udiNotificationClass := 22           );
  C_5640_501_06_RTC01_SPV_R0426_2 : FbAnalogValue_Medium (54) := (                _sDescription := 'Arbeidende settpunkt',                 _rCov_Increment := 0.1,                 _eUnits := WagoTypesBacnet.eBACnetUnits.UNIT_DEGREES_C           );
  C_5640_501_06_RTC01_SPV_Komf_R0426_2 : FbAnalogValue_Medium (55) := (                _sDescription := 'Settpunkt komfort',                 _rCov_Increment := 0.1,                 _eUnits := WagoTypesBacnet.eBACnetUnits.UNIT_DEGREES_C           );
  C_5640_501_06_RTC01_SPV_Stdb_R0426_2 : FbAnalogValue_Medium (56) := (                _sDescription := 'Settpunkt Standby',                 _rCov_Increment := 0.1,                 _eUnits := WagoTypesBacnet.eBACnetUnits.UNIT_DEGREES_C           );
  C_5640_501_06_RTC01_SPV_Natt_R0426_2 : FbAnalogValue_Medium (57) := (                _sDescription := 'Settpunkt Natt',                 _rCov_Increment := 0.1,                 _eUnits := WagoTypesBacnet.eBACnetUnits.UNIT_DEGREES_C           );
  C_5640_501_06_RTC01_MOD_FB_R0426_2 : FbMultiStateValue_Large (18) := (                _sDescription := 'Tilbakemelding driftmodus',                 _udiNumberOfStates := 5,                 _xEventDetectionEnable := FALSE,                 _udiNotificationClass := 99           );
  C_5640_501_06_RTC01_KMD_MSV_R0426_2 : FbMultiStateValue_Large (19) := (                _sDescription := 'Kalender',                 _udiNumberOfStates := 10,                 _xEventDetectionEnable := FALSE,                 _udiNotificationClass := 99           );
  C_5640_501_06_RTC01_SP_Tid_Stdb_R0426_2 : FbAnalogValue_Medium (58) := (                _sDescription := 'Utløpstid tilstedeværelse',                 _rCov_Increment := 1,                 _eUnits := WagoTypesBacnet.eBACnetUnits.UNIT_MINUTES           );
  C_5640_501_06_RYA601_SP_R0426_2 : FbAnalogValue_Medium (59) := (                _sDescription := 'Settpunkt',                 _rCov_Increment := 1,                 _eUnits := WagoTypesBacnet.eBACnetUnits.UNIT_PARTS_PER_MILLION           );
  C_5640_501_06_RYA601_MV_R0426_2 : FbAnalogInput_Large (19) := (                _sDescription := 'Målt CO2-konsentrasjon',                 _rCov_Increment := 1,                 _eUnits := WagoTypesBacnet.eBACnetUnits.UNIT_PARTS_PER_MILLION,                 _rHighLimit := 1000,                 _ILimitEnable := ( xLowLimitReporting := FALSE, xHighLimitReporting := TRUE ),                 _udiNotificationClass := 22           );
  C_5640_501_06_SBB01_C_R0426_2 : FbAnalogOutput_Medium (9) := (                _sDescription := 'Pådrag varmeorgan',                 _rCov_Increment := 1,                 _eUnits := WagoTypesBacnet.eBACnetUnits.UNIT_PERCENT           );
  C_5640_501_06_RBA01_D_R0426_3 : FbBinaryOutput_Medium (10) := (                _sDescription := 'Tilstedeværelsesdetektor',                 _sActiveText := 'Tilstedeværelse',                 _sInactiveText := 'Ingen tilstedeværelse'           );
  C_5640_501_06_RTC01_MV_R0426_3 : FbAnalogInput_Large (20) := (                _sDescription := 'Målt temperatur',                 _rCov_Increment := 0.1,                 _eUnits := WagoTypesBacnet.eBACnetUnits.UNIT_DEGREES_C,                 _rHighLimit := 28,                 _ILimitEnable := ( xLowLimitReporting := FALSE, xHighLimitReporting := TRUE ),                 _udiNotificationClass := 22           );
  C_5640_501_06_RTC01_SPV_R0426_3 : FbAnalogValue_Medium (60) := (                _sDescription := 'Arbeidende settpunkt',                 _rCov_Increment := 0.1,                 _eUnits := WagoTypesBacnet.eBACnetUnits.UNIT_DEGREES_C           );
  C_5640_501_06_RTC01_SPV_Komf_R0426_3 : FbAnalogValue_Medium (61) := (                _sDescription := 'Settpunkt komfort',                 _rCov_Increment := 0.1,                 _eUnits := WagoTypesBacnet.eBACnetUnits.UNIT_DEGREES_C           );
  C_5640_501_06_RTC01_SPV_Stdb_R0426_3 : FbAnalogValue_Medium (62) := (                _sDescription := 'Settpunkt Standby',                 _rCov_Increment := 0.1,                 _eUnits := WagoTypesBacnet.eBACnetUnits.UNIT_DEGREES_C           );
  C_5640_501_06_RTC01_SPV_Natt_R0426_3 : FbAnalogValue_Medium (63) := (                _sDescription := 'Settpunkt Natt',                 _rCov_Increment := 0.1,                 _eUnits := WagoTypesBacnet.eBACnetUnits.UNIT_DEGREES_C           );
  C_5640_501_06_RTC01_MOD_FB_R0426_3 : FbMultiStateValue_Large (20) := (                _sDescription := 'Tilbakemelding driftmodus',                 _udiNumberOfStates := 5,                 _xEventDetectionEnable := FALSE,                 _udiNotificationClass := 99           );
  C_5640_501_06_RTC01_KMD_MSV_R0426_3 : FbMultiStateValue_Large (21) := (                _sDescription := 'Kalender',                 _udiNumberOfStates := 10,                 _xEventDetectionEnable := FALSE,                 _udiNotificationClass := 99           );
  C_5640_501_06_RTC01_SP_Tid_Stdb_R0426_3 : FbAnalogValue_Medium (64) := (                _sDescription := 'Utløpstid tilstedeværelse',                 _rCov_Increment := 1,                 _eUnits := WagoTypesBacnet.eBACnetUnits.UNIT_MINUTES           );
  C_5640_501_06_RYA601_SP_R0426_3 : FbAnalogValue_Medium (65) := (                _sDescription := 'Settpunkt',                 _rCov_Increment := 1,                 _eUnits := WagoTypesBacnet.eBACnetUnits.UNIT_PARTS_PER_MILLION           );
  C_5640_501_06_RYA601_MV_R0426_3 : FbAnalogInput_Large (21) := (                _sDescription := 'Målt CO2-konsentrasjon',                 _rCov_Increment := 1,                 _eUnits := WagoTypesBacnet.eBACnetUnits.UNIT_PARTS_PER_MILLION,                 _rHighLimit := 1000,                 _ILimitEnable := ( xLowLimitReporting := FALSE, xHighLimitReporting := TRUE ),                 _udiNotificationClass := 22           );
  C_5640_501_06_SBB01_C_R0426_3 : FbAnalogOutput_Medium (10) := (                _sDescription := 'Pådrag varmeorgan',                 _rCov_Increment := 1,                 _eUnits := WagoTypesBacnet.eBACnetUnits.UNIT_PERCENT           );
  C_5640_501_06_RBA01_D_R0528 : FbBinaryOutput_Medium (11) := (                _sDescription := 'Tilstedeværelsesdetektor',                 _sActiveText := 'Tilstedeværelse',                 _sInactiveText := 'Ingen tilstedeværelse'           );
  C_5640_501_06_RTC01_MV_R0528 : FbAnalogInput_Large (22) := (                _sDescription := 'Målt temperatur',                 _rCov_Increment := 0.1,                 _eUnits := WagoTypesBacnet.eBACnetUnits.UNIT_DEGREES_C,                 _rHighLimit := 28,                 _ILimitEnable := ( xLowLimitReporting := FALSE, xHighLimitReporting := TRUE ),                 _udiNotificationClass := 22           );
  C_5640_501_06_RTC01_SPV_R0528 : FbAnalogValue_Medium (66) := (                _sDescription := 'Arbeidende settpunkt',                 _rCov_Increment := 0.1,                 _eUnits := WagoTypesBacnet.eBACnetUnits.UNIT_DEGREES_C           );
  C_5640_501_06_RTC01_SPV_Komf_R0528 : FbAnalogValue_Medium (67) := (                _sDescription := 'Settpunkt komfort',                 _rCov_Increment := 0.1,                 _eUnits := WagoTypesBacnet.eBACnetUnits.UNIT_DEGREES_C           );
  C_5640_501_06_RTC01_SPV_Stdb_R0528 : FbAnalogValue_Medium (68) := (                _sDescription := 'Settpunkt Standby',                 _rCov_Increment := 0.1,                 _eUnits := WagoTypesBacnet.eBACnetUnits.UNIT_DEGREES_C           );
  C_5640_501_06_RTC01_SPV_Natt_R0528 : FbAnalogValue_Medium (69) := (                _sDescription := 'Settpunkt Natt',                 _rCov_Increment := 0.1,                 _eUnits := WagoTypesBacnet.eBACnetUnits.UNIT_DEGREES_C           );
  C_5640_501_06_RTC01_MOD_FB_R0528 : FbMultiStateValue_Large (22) := (                _sDescription := 'Tilbakemelding driftmodus',                 _udiNumberOfStates := 5,                 _xEventDetectionEnable := FALSE,                 _udiNotificationClass := 99           );
  C_5640_501_06_RTC01_KMD_MSV_R0528 : FbMultiStateValue_Large (23) := (                _sDescription := 'Kalender',                 _udiNumberOfStates := 10,                 _xEventDetectionEnable := FALSE,                 _udiNotificationClass := 99           );
  C_5640_501_06_RTC01_SP_Tid_Stdb_R0528 : FbAnalogValue_Medium (70) := (                _sDescription := 'Utløpstid tilstedeværelse',                 _rCov_Increment := 1,                 _eUnits := WagoTypesBacnet.eBACnetUnits.UNIT_MINUTES           );
  C_5640_501_06_RYA601_SP_R0528 : FbAnalogValue_Medium (71) := (                _sDescription := 'Settpunkt',                 _rCov_Increment := 1,                 _eUnits := WagoTypesBacnet.eBACnetUnits.UNIT_PARTS_PER_MILLION           );
  C_5640_501_06_RYA601_MV_R0528 : FbAnalogInput_Large (23) := (                _sDescription := 'Målt CO2-konsentrasjon',                 _rCov_Increment := 1,                 _eUnits := WagoTypesBacnet.eBACnetUnits.UNIT_PARTS_PER_MILLION,                 _rHighLimit := 1000,                 _ILimitEnable := ( xLowLimitReporting := FALSE, xHighLimitReporting := TRUE ),                 _udiNotificationClass := 22           );
  C_5640_501_06_SBB01_C_R0528 : FbAnalogOutput_Medium (11) := (                _sDescription := 'Pådrag varmeorgan',                 _rCov_Increment := 1,                 _eUnits := WagoTypesBacnet.eBACnetUnits.UNIT_PERCENT           );
  C_5640_501_06_RBA01_D_R0523 : FbBinaryOutput_Medium (12) := (                _sDescription := 'Tilstedeværelsesdetektor',                 _sActiveText := 'Tilstedeværelse',                 _sInactiveText := 'Ingen tilstedeværelse'           );
  C_5640_501_06_RTC01_MV_R0523 : FbAnalogInput_Large (24) := (                _sDescription := 'Målt temperatur',                 _rCov_Increment := 0.1,                 _eUnits := WagoTypesBacnet.eBACnetUnits.UNIT_DEGREES_C,                 _rHighLimit := 28,                 _ILimitEnable := ( xLowLimitReporting := FALSE, xHighLimitReporting := TRUE ),                 _udiNotificationClass := 22           );
  C_5640_501_06_RTC01_SPV_R0523 : FbAnalogValue_Medium (72) := (                _sDescription := 'Arbeidende settpunkt',                 _rCov_Increment := 0.1,                 _eUnits := WagoTypesBacnet.eBACnetUnits.UNIT_DEGREES_C           );
  C_5640_501_06_RTC01_SPV_Komf_R0523 : FbAnalogValue_Medium (73) := (                _sDescription := 'Settpunkt komfort',                 _rCov_Increment := 0.1,                 _eUnits := WagoTypesBacnet.eBACnetUnits.UNIT_DEGREES_C           );
  C_5640_501_06_RTC01_SPV_Stdb_R0523 : FbAnalogValue_Medium (74) := (                _sDescription := 'Settpunkt Standby',                 _rCov_Increment := 0.1,                 _eUnits := WagoTypesBacnet.eBACnetUnits.UNIT_DEGREES_C           );
  C_5640_501_06_RTC01_SPV_Natt_R0523 : FbAnalogValue_Medium (75) := (                _sDescription := 'Settpunkt Natt',                 _rCov_Increment := 0.1,                 _eUnits := WagoTypesBacnet.eBACnetUnits.UNIT_DEGREES_C           );
  C_5640_501_06_RTC01_MOD_FB_R0523 : FbMultiStateValue_Large (24) := (                _sDescription := 'Tilbakemelding driftmodus',                 _udiNumberOfStates := 5,                 _xEventDetectionEnable := FALSE,                 _udiNotificationClass := 99           );
  C_5640_501_06_RTC01_KMD_MSV_R0523 : FbMultiStateValue_Large (25) := (                _sDescription := 'Kalender',                 _udiNumberOfStates := 10,                 _xEventDetectionEnable := FALSE,                 _udiNotificationClass := 99           );
  C_5640_501_06_RTC01_SP_Tid_Stdb_R0523 : FbAnalogValue_Medium (76) := (                _sDescription := 'Utløpstid tilstedeværelse',                 _rCov_Increment := 1,                 _eUnits := WagoTypesBacnet.eBACnetUnits.UNIT_MINUTES           );
  C_5640_501_06_RYA601_SP_R0523 : FbAnalogValue_Medium (77) := (                _sDescription := 'Settpunkt',                 _rCov_Increment := 1,                 _eUnits := WagoTypesBacnet.eBACnetUnits.UNIT_PARTS_PER_MILLION           );
  C_5640_501_06_RYA601_MV_R0523 : FbAnalogInput_Large (25) := (                _sDescription := 'Målt CO2-konsentrasjon',                 _rCov_Increment := 1,                 _eUnits := WagoTypesBacnet.eBACnetUnits.UNIT_PARTS_PER_MILLION,                 _rHighLimit := 1000,                 _ILimitEnable := ( xLowLimitReporting := FALSE, xHighLimitReporting := TRUE ),                 _udiNotificationClass := 22           );
  C_5640_501_06_SBB01_C_R0523 : FbAnalogOutput_Medium (12) := (                _sDescription := 'Pådrag varmeorgan',                 _rCov_Increment := 1,                 _eUnits := WagoTypesBacnet.eBACnetUnits.UNIT_PERCENT           );
  C_5640_501_06_RBA01_D_R0531 : FbBinaryOutput_Medium (13) := (                _sDescription := 'Tilstedeværelsesdetektor',                 _sActiveText := 'Tilstedeværelse',                 _sInactiveText := 'Ingen tilstedeværelse'           );
  C_5640_501_06_RTC01_MV_R0531 : FbAnalogInput_Large (26) := (                _sDescription := 'Målt temperatur',                 _rCov_Increment := 0.1,                 _eUnits := WagoTypesBacnet.eBACnetUnits.UNIT_DEGREES_C,                 _rHighLimit := 28,                 _ILimitEnable := ( xLowLimitReporting := FALSE, xHighLimitReporting := TRUE ),                 _udiNotificationClass := 22           );
  C_5640_501_06_RTC01_SPV_R0531 : FbAnalogValue_Medium (78) := (                _sDescription := 'Arbeidende settpunkt',                 _rCov_Increment := 0.1,                 _eUnits := WagoTypesBacnet.eBACnetUnits.UNIT_DEGREES_C           );
  C_5640_501_06_RTC01_SPV_Komf_R0531 : FbAnalogValue_Medium (79) := (                _sDescription := 'Settpunkt komfort',                 _rCov_Increment := 0.1,                 _eUnits := WagoTypesBacnet.eBACnetUnits.UNIT_DEGREES_C           );
  C_5640_501_06_RTC01_SPV_Stdb_R0531 : FbAnalogValue_Medium (80) := (                _sDescription := 'Settpunkt Standby',                 _rCov_Increment := 0.1,                 _eUnits := WagoTypesBacnet.eBACnetUnits.UNIT_DEGREES_C           );
  C_5640_501_06_RTC01_SPV_Natt_R0531 : FbAnalogValue_Medium (81) := (                _sDescription := 'Settpunkt Natt',                 _rCov_Increment := 0.1,                 _eUnits := WagoTypesBacnet.eBACnetUnits.UNIT_DEGREES_C           );
  C_5640_501_06_RTC01_MOD_FB_R0531 : FbMultiStateValue_Large (26) := (                _sDescription := 'Tilbakemelding driftmodus',                 _udiNumberOfStates := 5,                 _xEventDetectionEnable := FALSE,                 _udiNotificationClass := 99           );
  C_5640_501_06_RTC01_KMD_MSV_R0531 : FbMultiStateValue_Large (27) := (                _sDescription := 'Kalender',                 _udiNumberOfStates := 10,                 _xEventDetectionEnable := FALSE,                 _udiNotificationClass := 99           );
  C_5640_501_06_RTC01_SP_Tid_Stdb_R0531 : FbAnalogValue_Medium (82) := (                _sDescription := 'Utløpstid tilstedeværelse',                 _rCov_Increment := 1,                 _eUnits := WagoTypesBacnet.eBACnetUnits.UNIT_MINUTES           );
  C_5640_501_06_RYA601_SP_R0531 : FbAnalogValue_Medium (83) := (                _sDescription := 'Settpunkt',                 _rCov_Increment := 1,                 _eUnits := WagoTypesBacnet.eBACnetUnits.UNIT_PARTS_PER_MILLION           );
  C_5640_501_06_RYA601_MV_R0531 : FbAnalogInput_Large (27) := (                _sDescription := 'Målt CO2-konsentrasjon',                 _rCov_Increment := 1,                 _eUnits := WagoTypesBacnet.eBACnetUnits.UNIT_PARTS_PER_MILLION,                 _rHighLimit := 1000,                 _ILimitEnable := ( xLowLimitReporting := FALSE, xHighLimitReporting := TRUE ),                 _udiNotificationClass := 22           );
  C_5640_501_06_SBB01_C_R0531 : FbAnalogOutput_Medium (13) := (                _sDescription := 'Pådrag varmeorgan',                 _rCov_Increment := 1,                 _eUnits := WagoTypesBacnet.eBACnetUnits.UNIT_PERCENT           );
  C_5640_501_06_RBA01_D_R0535_1 : FbBinaryOutput_Medium (14) := (                _sDescription := 'Tilstedeværelsesdetektor',                 _sActiveText := 'Tilstedeværelse',                 _sInactiveText := 'Ingen tilstedeværelse'           );
  C_5640_501_06_RTC01_MV_R0535_1 : FbAnalogInput_Large (28) := (                _sDescription := 'Målt temperatur',                 _rCov_Increment := 0.1,                 _eUnits := WagoTypesBacnet.eBACnetUnits.UNIT_DEGREES_C,                 _rHighLimit := 28,                 _ILimitEnable := ( xLowLimitReporting := FALSE, xHighLimitReporting := TRUE ),                 _udiNotificationClass := 22           );
  C_5640_501_06_RTC01_SPV_R0535_1 : FbAnalogValue_Medium (84) := (                _sDescription := 'Arbeidende settpunkt',                 _rCov_Increment := 0.1,                 _eUnits := WagoTypesBacnet.eBACnetUnits.UNIT_DEGREES_C           );
  C_5640_501_06_RTC01_SPV_Komf_R0535_1 : FbAnalogValue_Medium (85) := (                _sDescription := 'Settpunkt komfort',                 _rCov_Increment := 0.1,                 _eUnits := WagoTypesBacnet.eBACnetUnits.UNIT_DEGREES_C           );
  C_5640_501_06_RTC01_SPV_Stdb_R0535_1 : FbAnalogValue_Medium (86) := (                _sDescription := 'Settpunkt Standby',                 _rCov_Increment := 0.1,                 _eUnits := WagoTypesBacnet.eBACnetUnits.UNIT_DEGREES_C           );
  C_5640_501_06_RTC01_SPV_Natt_R0535_1 : FbAnalogValue_Medium (87) := (                _sDescription := 'Settpunkt Natt',                 _rCov_Increment := 0.1,                 _eUnits := WagoTypesBacnet.eBACnetUnits.UNIT_DEGREES_C           );
  C_5640_501_06_RTC01_MOD_FB_R0535_1 : FbMultiStateValue_Large (28) := (                _sDescription := 'Tilbakemelding driftmodus',                 _udiNumberOfStates := 5,                 _xEventDetectionEnable := FALSE,                 _udiNotificationClass := 99           );
  C_5640_501_06_RTC01_KMD_MSV_R0535_1 : FbMultiStateValue_Large (29) := (                _sDescription := 'Kalender',                 _udiNumberOfStates := 10,                 _xEventDetectionEnable := FALSE,                 _udiNotificationClass := 99           );
  C_5640_501_06_RTC01_SP_Tid_Stdb_R0535_1 : FbAnalogValue_Medium (88) := (                _sDescription := 'Utløpstid tilstedeværelse',                 _rCov_Increment := 1,                 _eUnits := WagoTypesBacnet.eBACnetUnits.UNIT_MINUTES           );
  C_5640_501_06_RYA601_SP_R0535_1 : FbAnalogValue_Medium (89) := (                _sDescription := 'Settpunkt',                 _rCov_Increment := 1,                 _eUnits := WagoTypesBacnet.eBACnetUnits.UNIT_PARTS_PER_MILLION           );
  C_5640_501_06_RYA601_MV_R0535_1 : FbAnalogInput_Large (29) := (                _sDescription := 'Målt CO2-konsentrasjon',                 _rCov_Increment := 1,                 _eUnits := WagoTypesBacnet.eBACnetUnits.UNIT_PARTS_PER_MILLION,                 _rHighLimit := 1000,                 _ILimitEnable := ( xLowLimitReporting := FALSE, xHighLimitReporting := TRUE ),                 _udiNotificationClass := 22           );
  C_5640_501_06_SBB01_C_R0535_1 : FbAnalogOutput_Medium (14) := (                _sDescription := 'Pådrag varmeorgan',                 _rCov_Increment := 1,                 _eUnits := WagoTypesBacnet.eBACnetUnits.UNIT_PERCENT           );
  C_5640_501_06_RBA01_D_R0535_2 : FbBinaryOutput_Medium (15) := (                _sDescription := 'Tilstedeværelsesdetektor',                 _sActiveText := 'Tilstedeværelse',                 _sInactiveText := 'Ingen tilstedeværelse'           );
  C_5640_501_06_RTC01_MV_R0535_2 : FbAnalogInput_Large (30) := (                _sDescription := 'Målt temperatur',                 _rCov_Increment := 0.1,                 _eUnits := WagoTypesBacnet.eBACnetUnits.UNIT_DEGREES_C,                 _rHighLimit := 28,                 _ILimitEnable := ( xLowLimitReporting := FALSE, xHighLimitReporting := TRUE ),                 _udiNotificationClass := 22           );
  C_5640_501_06_RTC01_SPV_R0535_2 : FbAnalogValue_Medium (90) := (                _sDescription := 'Arbeidende settpunkt',                 _rCov_Increment := 0.1,                 _eUnits := WagoTypesBacnet.eBACnetUnits.UNIT_DEGREES_C           );
  C_5640_501_06_RTC01_SPV_Komf_R0535_2 : FbAnalogValue_Medium (91) := (                _sDescription := 'Settpunkt komfort',                 _rCov_Increment := 0.1,                 _eUnits := WagoTypesBacnet.eBACnetUnits.UNIT_DEGREES_C           );
  C_5640_501_06_RTC01_SPV_Stdb_R0535_2 : FbAnalogValue_Medium (92) := (                _sDescription := 'Settpunkt Standby',                 _rCov_Increment := 0.1,                 _eUnits := WagoTypesBacnet.eBACnetUnits.UNIT_DEGREES_C           );
  C_5640_501_06_RTC01_SPV_Natt_R0535_2 : FbAnalogValue_Medium (93) := (                _sDescription := 'Settpunkt Natt',                 _rCov_Increment := 0.1,                 _eUnits := WagoTypesBacnet.eBACnetUnits.UNIT_DEGREES_C           );
  C_5640_501_06_RTC01_MOD_FB_R0535_2 : FbMultiStateValue_Large (30) := (                _sDescription := 'Tilbakemelding driftmodus',                 _udiNumberOfStates := 5,                 _xEventDetectionEnable := FALSE,                 _udiNotificationClass := 99           );
  C_5640_501_06_RTC01_KMD_MSV_R0535_2 : FbMultiStateValue_Large (31) := (                _sDescription := 'Kalender',                 _udiNumberOfStates := 10,                 _xEventDetectionEnable := FALSE,                 _udiNotificationClass := 99           );
  C_5640_501_06_RTC01_SP_Tid_Stdb_R0535_2 : FbAnalogValue_Medium (94) := (                _sDescription := 'Utløpstid tilstedeværelse',                 _rCov_Increment := 1,                 _eUnits := WagoTypesBacnet.eBACnetUnits.UNIT_MINUTES           );
  C_5640_501_06_RYA601_SP_R0535_2 : FbAnalogValue_Medium (95) := (                _sDescription := 'Settpunkt',                 _rCov_Increment := 1,                 _eUnits := WagoTypesBacnet.eBACnetUnits.UNIT_PARTS_PER_MILLION           );
  C_5640_501_06_RYA601_MV_R0535_2 : FbAnalogInput_Large (31) := (                _sDescription := 'Målt CO2-konsentrasjon',                 _rCov_Increment := 1,                 _eUnits := WagoTypesBacnet.eBACnetUnits.UNIT_PARTS_PER_MILLION,                 _rHighLimit := 1000,                 _ILimitEnable := ( xLowLimitReporting := FALSE, xHighLimitReporting := TRUE ),                 _udiNotificationClass := 22           );
  C_5640_501_06_SBB01_C_R0535_2 : FbAnalogOutput_Medium (15) := (                _sDescription := 'Pådrag varmeorgan',                 _rCov_Increment := 1,                 _eUnits := WagoTypesBacnet.eBACnetUnits.UNIT_PERCENT           );
  C_5640_501_06_RBA01_D_R0535_3 : FbBinaryOutput_Medium (16) := (                _sDescription := 'Tilstedeværelsesdetektor',                 _sActiveText := 'Tilstedeværelse',                 _sInactiveText := 'Ingen tilstedeværelse'           );
  C_5640_501_06_RTC01_MV_R0535_3 : FbAnalogInput_Large (32) := (                _sDescription := 'Målt temperatur',                 _rCov_Increment := 0.1,                 _eUnits := WagoTypesBacnet.eBACnetUnits.UNIT_DEGREES_C,                 _rHighLimit := 28,                 _ILimitEnable := ( xLowLimitReporting := FALSE, xHighLimitReporting := TRUE ),                 _udiNotificationClass := 22           );
  C_5640_501_06_RTC01_SPV_R0535_3 : FbAnalogValue_Medium (96) := (                _sDescription := 'Arbeidende settpunkt',                 _rCov_Increment := 0.1,                 _eUnits := WagoTypesBacnet.eBACnetUnits.UNIT_DEGREES_C           );
  C_5640_501_06_RTC01_SPV_Komf_R0535_3 : FbAnalogValue_Medium (97) := (                _sDescription := 'Settpunkt komfort',                 _rCov_Increment := 0.1,                 _eUnits := WagoTypesBacnet.eBACnetUnits.UNIT_DEGREES_C           );
  C_5640_501_06_RTC01_SPV_Stdb_R0535_3 : FbAnalogValue_Medium (98) := (                _sDescription := 'Settpunkt Standby',                 _rCov_Increment := 0.1,                 _eUnits := WagoTypesBacnet.eBACnetUnits.UNIT_DEGREES_C           );
  C_5640_501_06_RTC01_SPV_Natt_R0535_3 : FbAnalogValue_Medium (99) := (                _sDescription := 'Settpunkt Natt',                 _rCov_Increment := 0.1,                 _eUnits := WagoTypesBacnet.eBACnetUnits.UNIT_DEGREES_C           );
  C_5640_501_06_RTC01_MOD_FB_R0535_3 : FbMultiStateValue_Large (32) := (                _sDescription := 'Tilbakemelding driftmodus',                 _udiNumberOfStates := 5,                 _xEventDetectionEnable := FALSE,                 _udiNotificationClass := 99           );
  C_5640_501_06_RTC01_KMD_MSV_R0535_3 : FbMultiStateValue_Large (33) := (                _sDescription := 'Kalender',                 _udiNumberOfStates := 10,                 _xEventDetectionEnable := FALSE,                 _udiNotificationClass := 99           );
  C_5640_501_06_RTC01_SP_Tid_Stdb_R0535_3 : FbAnalogValue_Medium (100) := (                _sDescription := 'Utløpstid tilstedeværelse',                 _rCov_Increment := 1,                 _eUnits := WagoTypesBacnet.eBACnetUnits.UNIT_MINUTES           );
  C_5640_501_06_RYA601_SP_R0535_3 : FbAnalogValue_Medium (101) := (                _sDescription := 'Settpunkt',                 _rCov_Increment := 1,                 _eUnits := WagoTypesBacnet.eBACnetUnits.UNIT_PARTS_PER_MILLION           );
  C_5640_501_06_RYA601_MV_R0535_3 : FbAnalogInput_Large (33) := (                _sDescription := 'Målt CO2-konsentrasjon',                 _rCov_Increment := 1,                 _eUnits := WagoTypesBacnet.eBACnetUnits.UNIT_PARTS_PER_MILLION,                 _rHighLimit := 1000,                 _ILimitEnable := ( xLowLimitReporting := FALSE, xHighLimitReporting := TRUE ),                 _udiNotificationClass := 22           );
  C_5640_501_06_SBB01_C_R0535_3 : FbAnalogOutput_Medium (16) := (                _sDescription := 'Pådrag varmeorgan',                 _rCov_Increment := 1,                 _eUnits := WagoTypesBacnet.eBACnetUnits.UNIT_PERCENT           );
  C_5640_501_06_RBA01_D_R0536 : FbBinaryOutput_Medium (17) := (                _sDescription := 'Tilstedeværelsesdetektor',                 _sActiveText := 'Tilstedeværelse',                 _sInactiveText := 'Ingen tilstedeværelse'           );
  C_5640_501_06_RTC01_MV_R0536 : FbAnalogInput_Large (34) := (                _sDescription := 'Målt temperatur',                 _rCov_Increment := 0.1,                 _eUnits := WagoTypesBacnet.eBACnetUnits.UNIT_DEGREES_C,                 _rHighLimit := 28,                 _ILimitEnable := ( xLowLimitReporting := FALSE, xHighLimitReporting := TRUE ),                 _udiNotificationClass := 22           );
  C_5640_501_06_RTC01_SPV_R0536 : FbAnalogValue_Medium (102) := (                _sDescription := 'Arbeidende settpunkt',                 _rCov_Increment := 0.1,                 _eUnits := WagoTypesBacnet.eBACnetUnits.UNIT_DEGREES_C           );
  C_5640_501_06_RTC01_SPV_Komf_R0536 : FbAnalogValue_Medium (103) := (                _sDescription := 'Settpunkt komfort',                 _rCov_Increment := 0.1,                 _eUnits := WagoTypesBacnet.eBACnetUnits.UNIT_DEGREES_C           );
  C_5640_501_06_RTC01_SPV_Stdb_R0536 : FbAnalogValue_Medium (104) := (                _sDescription := 'Settpunkt Standby',                 _rCov_Increment := 0.1,                 _eUnits := WagoTypesBacnet.eBACnetUnits.UNIT_DEGREES_C           );
  C_5640_501_06_RTC01_SPV_Natt_R0536 : FbAnalogValue_Medium (105) := (                _sDescription := 'Settpunkt Natt',                 _rCov_Increment := 0.1,                 _eUnits := WagoTypesBacnet.eBACnetUnits.UNIT_DEGREES_C           );
  C_5640_501_06_RTC01_MOD_FB_R0536 : FbMultiStateValue_Large (34) := (                _sDescription := 'Tilbakemelding driftmodus',                 _udiNumberOfStates := 5,                 _xEventDetectionEnable := FALSE,                 _udiNotificationClass := 99           );
  C_5640_501_06_RTC01_KMD_MSV_R0536 : FbMultiStateValue_Large (35) := (                _sDescription := 'Kalender',                 _udiNumberOfStates := 10,                 _xEventDetectionEnable := FALSE,                 _udiNotificationClass := 99           );
  C_5640_501_06_RTC01_SP_Tid_Stdb_R0536 : FbAnalogValue_Medium (106) := (                _sDescription := 'Utløpstid tilstedeværelse',                 _rCov_Increment := 1,                 _eUnits := WagoTypesBacnet.eBACnetUnits.UNIT_MINUTES           );
  C_5640_501_06_RYA601_SP_R0536 : FbAnalogValue_Medium (107) := (                _sDescription := 'Settpunkt',                 _rCov_Increment := 1,                 _eUnits := WagoTypesBacnet.eBACnetUnits.UNIT_PARTS_PER_MILLION           );
  C_5640_501_06_RYA601_MV_R0536 : FbAnalogInput_Large (35) := (                _sDescription := 'Målt CO2-konsentrasjon',                 _rCov_Increment := 1,                 _eUnits := WagoTypesBacnet.eBACnetUnits.UNIT_PARTS_PER_MILLION,                 _rHighLimit := 1000,                 _ILimitEnable := ( xLowLimitReporting := FALSE, xHighLimitReporting := TRUE ),                 _udiNotificationClass := 22           );
  C_5640_501_06_SBB01_C_R0536 : FbAnalogOutput_Medium (17) := (                _sDescription := 'Pådrag varmeorgan',                 _rCov_Increment := 1,                 _eUnits := WagoTypesBacnet.eBACnetUnits.UNIT_PERCENT           );
  C_5640_501_06_RBA01_D_R0543 : FbBinaryOutput_Medium (18) := (                _sDescription := 'Tilstedeværelsesdetektor',                 _sActiveText := 'Tilstedeværelse',                 _sInactiveText := 'Ingen tilstedeværelse'           );
  C_5640_501_06_RTC01_MV_R0543 : FbAnalogInput_Large (36) := (                _sDescription := 'Målt temperatur',                 _rCov_Increment := 0.1,                 _eUnits := WagoTypesBacnet.eBACnetUnits.UNIT_DEGREES_C,                 _rHighLimit := 28,                 _ILimitEnable := ( xLowLimitReporting := FALSE, xHighLimitReporting := TRUE ),                 _udiNotificationClass := 22           );
  C_5640_501_06_RTC01_SPV_R0543 : FbAnalogValue_Medium (108) := (                _sDescription := 'Arbeidende settpunkt',                 _rCov_Increment := 0.1,                 _eUnits := WagoTypesBacnet.eBACnetUnits.UNIT_DEGREES_C           );
  C_5640_501_06_RTC01_SPV_Komf_R0543 : FbAnalogValue_Medium (109) := (                _sDescription := 'Settpunkt komfort',                 _rCov_Increment := 0.1,                 _eUnits := WagoTypesBacnet.eBACnetUnits.UNIT_DEGREES_C           );
  C_5640_501_06_RTC01_SPV_Stdb_R0543 : FbAnalogValue_Medium (110) := (                _sDescription := 'Settpunkt Standby',                 _rCov_Increment := 0.1,                 _eUnits := WagoTypesBacnet.eBACnetUnits.UNIT_DEGREES_C           );
  C_5640_501_06_RTC01_SPV_Natt_R0543 : FbAnalogValue_Medium (111) := (                _sDescription := 'Settpunkt Natt',                 _rCov_Increment := 0.1,                 _eUnits := WagoTypesBacnet.eBACnetUnits.UNIT_DEGREES_C           );
  C_5640_501_06_RTC01_MOD_FB_R0543 : FbMultiStateValue_Large (36) := (                _sDescription := 'Tilbakemelding driftmodus',                 _udiNumberOfStates := 5,                 _xEventDetectionEnable := FALSE,                 _udiNotificationClass := 99           );
  C_5640_501_06_RTC01_KMD_MSV_R0543 : FbMultiStateValue_Large (37) := (                _sDescription := 'Kalender',                 _udiNumberOfStates := 10,                 _xEventDetectionEnable := FALSE,                 _udiNotificationClass := 99           );
  C_5640_501_06_RTC01_SP_Tid_Stdb_R0543 : FbAnalogValue_Medium (112) := (                _sDescription := 'Utløpstid tilstedeværelse',                 _rCov_Increment := 1,                 _eUnits := WagoTypesBacnet.eBACnetUnits.UNIT_MINUTES           );
  C_5640_501_06_RYA601_SP_R0543 : FbAnalogValue_Medium (113) := (                _sDescription := 'Settpunkt',                 _rCov_Increment := 1,                 _eUnits := WagoTypesBacnet.eBACnetUnits.UNIT_PARTS_PER_MILLION           );
  C_5640_501_06_RYA601_MV_R0543 : FbAnalogInput_Large (37) := (                _sDescription := 'Målt CO2-konsentrasjon',                 _rCov_Increment := 1,                 _eUnits := WagoTypesBacnet.eBACnetUnits.UNIT_PARTS_PER_MILLION,                 _rHighLimit := 1000,                 _ILimitEnable := ( xLowLimitReporting := FALSE, xHighLimitReporting := TRUE ),                 _udiNotificationClass := 22           );
  C_5640_501_06_SBB01_C_R0543 : FbAnalogOutput_Medium (18) := (                _sDescription := 'Pådrag varmeorgan',                 _rCov_Increment := 1,                 _eUnits := WagoTypesBacnet.eBACnetUnits.UNIT_PERCENT           );
  C_5640_501_06_RBA01_D_R0547_1 : FbBinaryOutput_Medium (19) := (                _sDescription := 'Tilstedeværelsesdetektor',                 _sActiveText := 'Tilstedeværelse',                 _sInactiveText := 'Ingen tilstedeværelse'           );
  C_5640_501_06_RTC01_MV_R0547_1 : FbAnalogInput_Large (38) := (                _sDescription := 'Målt temperatur',                 _rCov_Increment := 0.1,                 _eUnits := WagoTypesBacnet.eBACnetUnits.UNIT_DEGREES_C,                 _rHighLimit := 28,                 _ILimitEnable := ( xLowLimitReporting := FALSE, xHighLimitReporting := TRUE ),                 _udiNotificationClass := 22           );
  C_5640_501_06_RTC01_SPV_R0547_1 : FbAnalogValue_Medium (114) := (                _sDescription := 'Arbeidende settpunkt',                 _rCov_Increment := 0.1,                 _eUnits := WagoTypesBacnet.eBACnetUnits.UNIT_DEGREES_C           );
  C_5640_501_06_RTC01_SPV_Komf_R0547_1 : FbAnalogValue_Medium (115) := (                _sDescription := 'Settpunkt komfort',                 _rCov_Increment := 0.1,                 _eUnits := WagoTypesBacnet.eBACnetUnits.UNIT_DEGREES_C           );
  C_5640_501_06_RTC01_SPV_Stdb_R0547_1 : FbAnalogValue_Medium (116) := (                _sDescription := 'Settpunkt Standby',                 _rCov_Increment := 0.1,                 _eUnits := WagoTypesBacnet.eBACnetUnits.UNIT_DEGREES_C           );
  C_5640_501_06_RTC01_SPV_Natt_R0547_1 : FbAnalogValue_Medium (117) := (                _sDescription := 'Settpunkt Natt',                 _rCov_Increment := 0.1,                 _eUnits := WagoTypesBacnet.eBACnetUnits.UNIT_DEGREES_C           );
  C_5640_501_06_RTC01_MOD_FB_R0547_1 : FbMultiStateValue_Large (38) := (                _sDescription := 'Tilbakemelding driftmodus',                 _udiNumberOfStates := 5,                 _xEventDetectionEnable := FALSE,                 _udiNotificationClass := 99           );
  C_5640_501_06_RTC01_KMD_MSV_R0547_1 : FbMultiStateValue_Large (39) := (                _sDescription := 'Kalender',                 _udiNumberOfStates := 10,                 _xEventDetectionEnable := FALSE,                 _udiNotificationClass := 99           );
  C_5640_501_06_RTC01_SP_Tid_Stdb_R0547_1 : FbAnalogValue_Medium (118) := (                _sDescription := 'Utløpstid tilstedeværelse',                 _rCov_Increment := 1,                 _eUnits := WagoTypesBacnet.eBACnetUnits.UNIT_MINUTES           );
  C_5640_501_06_RYA601_SP_R0547_1 : FbAnalogValue_Medium (119) := (                _sDescription := 'Settpunkt',                 _rCov_Increment := 1,                 _eUnits := WagoTypesBacnet.eBACnetUnits.UNIT_PARTS_PER_MILLION           );
  C_5640_501_06_RYA601_MV_R0547_1 : FbAnalogInput_Large (39) := (                _sDescription := 'Målt CO2-konsentrasjon',                 _rCov_Increment := 1,                 _eUnits := WagoTypesBacnet.eBACnetUnits.UNIT_PARTS_PER_MILLION,                 _rHighLimit := 1000,                 _ILimitEnable := ( xLowLimitReporting := FALSE, xHighLimitReporting := TRUE ),                 _udiNotificationClass := 22           );
  C_5640_501_06_SBB01_C_R0547_1 : FbAnalogOutput_Medium (19) := (                _sDescription := 'Pådrag varmeorgan',                 _rCov_Increment := 1,                 _eUnits := WagoTypesBacnet.eBACnetUnits.UNIT_PERCENT           );
  C_5640_501_06_RBA01_D_R0547_2 : FbBinaryOutput_Medium (20) := (                _sDescription := 'Tilstedeværelsesdetektor',                 _sActiveText := 'Tilstedeværelse',                 _sInactiveText := 'Ingen tilstedeværelse'           );
  C_5640_501_06_RTC01_MV_R0547_2 : FbAnalogInput_Large (40) := (                _sDescription := 'Målt temperatur',                 _rCov_Increment := 0.1,                 _eUnits := WagoTypesBacnet.eBACnetUnits.UNIT_DEGREES_C,                 _rHighLimit := 28,                 _ILimitEnable := ( xLowLimitReporting := FALSE, xHighLimitReporting := TRUE ),                 _udiNotificationClass := 22           );
  C_5640_501_06_RTC01_SPV_R0547_2 : FbAnalogValue_Medium (120) := (                _sDescription := 'Arbeidende settpunkt',                 _rCov_Increment := 0.1,                 _eUnits := WagoTypesBacnet.eBACnetUnits.UNIT_DEGREES_C           );
  C_5640_501_06_RTC01_SPV_Komf_R0547_2 : FbAnalogValue_Medium (121) := (                _sDescription := 'Settpunkt komfort',                 _rCov_Increment := 0.1,                 _eUnits := WagoTypesBacnet.eBACnetUnits.UNIT_DEGREES_C           );
  C_5640_501_06_RTC01_SPV_Stdb_R0547_2 : FbAnalogValue_Medium (122) := (                _sDescription := 'Settpunkt Standby',                 _rCov_Increment := 0.1,                 _eUnits := WagoTypesBacnet.eBACnetUnits.UNIT_DEGREES_C           );
  C_5640_501_06_RTC01_SPV_Natt_R0547_2 : FbAnalogValue_Medium (123) := (                _sDescription := 'Settpunkt Natt',                 _rCov_Increment := 0.1,                 _eUnits := WagoTypesBacnet.eBACnetUnits.UNIT_DEGREES_C           );
  C_5640_501_06_RTC01_MOD_FB_R0547_2 : FbMultiStateValue_Large (40) := (                _sDescription := 'Tilbakemelding driftmodus',                 _udiNumberOfStates := 5,                 _xEventDetectionEnable := FALSE,                 _udiNotificationClass := 99           );
  C_5640_501_06_RTC01_KMD_MSV_R0547_2 : FbMultiStateValue_Large (41) := (                _sDescription := 'Kalender',                 _udiNumberOfStates := 10,                 _xEventDetectionEnable := FALSE,                 _udiNotificationClass := 99           );
  C_5640_501_06_RTC01_SP_Tid_Stdb_R0547_2 : FbAnalogValue_Medium (124) := (                _sDescription := 'Utløpstid tilstedeværelse',                 _rCov_Increment := 1,                 _eUnits := WagoTypesBacnet.eBACnetUnits.UNIT_MINUTES           );
  C_5640_501_06_RYA601_SP_R0547_2 : FbAnalogValue_Medium (125) := (                _sDescription := 'Settpunkt',                 _rCov_Increment := 1,                 _eUnits := WagoTypesBacnet.eBACnetUnits.UNIT_PARTS_PER_MILLION           );
  C_5640_501_06_RYA601_MV_R0547_2 : FbAnalogInput_Large (41) := (                _sDescription := 'Målt CO2-konsentrasjon',                 _rCov_Increment := 1,                 _eUnits := WagoTypesBacnet.eBACnetUnits.UNIT_PARTS_PER_MILLION,                 _rHighLimit := 1000,                 _ILimitEnable := ( xLowLimitReporting := FALSE, xHighLimitReporting := TRUE ),                 _udiNotificationClass := 22           );
  C_5640_501_06_SBB01_C_R0547_2 : FbAnalogOutput_Medium (20) := (                _sDescription := 'Pådrag varmeorgan',                 _rCov_Increment := 1,                 _eUnits := WagoTypesBacnet.eBACnetUnits.UNIT_PERCENT           );
  C_5640_501_06_RBA01_D_R0544 : FbBinaryOutput_Medium (21) := (                _sDescription := 'Tilstedeværelsesdetektor',                 _sActiveText := 'Tilstedeværelse',                 _sInactiveText := 'Ingen tilstedeværelse'           );
  C_5640_501_06_RTC01_MV_R0544 : FbAnalogInput_Large (42) := (                _sDescription := 'Målt temperatur',                 _rCov_Increment := 0.1,                 _eUnits := WagoTypesBacnet.eBACnetUnits.UNIT_DEGREES_C,                 _rHighLimit := 28,                 _ILimitEnable := ( xLowLimitReporting := FALSE, xHighLimitReporting := TRUE ),                 _udiNotificationClass := 22           );
  C_5640_501_06_RTC01_SPV_R0544 : FbAnalogValue_Medium (126) := (                _sDescription := 'Arbeidende settpunkt',                 _rCov_Increment := 0.1,                 _eUnits := WagoTypesBacnet.eBACnetUnits.UNIT_DEGREES_C           );
  C_5640_501_06_RTC01_SPV_Komf_R0544 : FbAnalogValue_Medium (127) := (                _sDescription := 'Settpunkt komfort',                 _rCov_Increment := 0.1,                 _eUnits := WagoTypesBacnet.eBACnetUnits.UNIT_DEGREES_C           );
  C_5640_501_06_RTC01_SPV_Stdb_R0544 : FbAnalogValue_Medium (128) := (                _sDescription := 'Settpunkt Standby',                 _rCov_Increment := 0.1,                 _eUnits := WagoTypesBacnet.eBACnetUnits.UNIT_DEGREES_C           );
  C_5640_501_06_RTC01_SPV_Natt_R0544 : FbAnalogValue_Medium (129) := (                _sDescription := 'Settpunkt Natt',                 _rCov_Increment := 0.1,                 _eUnits := WagoTypesBacnet.eBACnetUnits.UNIT_DEGREES_C           );
  C_5640_501_06_RTC01_MOD_FB_R0544 : FbMultiStateValue_Large (42) := (                _sDescription := 'Tilbakemelding driftmodus',                 _udiNumberOfStates := 5,                 _xEventDetectionEnable := FALSE,                 _udiNotificationClass := 99           );
  C_5640_501_06_RTC01_KMD_MSV_R0544 : FbMultiStateValue_Large (43) := (                _sDescription := 'Kalender',                 _udiNumberOfStates := 10,                 _xEventDetectionEnable := FALSE,                 _udiNotificationClass := 99           );
  C_5640_501_06_RTC01_SP_Tid_Stdb_R0544 : FbAnalogValue_Medium (130) := (                _sDescription := 'Utløpstid tilstedeværelse',                 _rCov_Increment := 1,                 _eUnits := WagoTypesBacnet.eBACnetUnits.UNIT_MINUTES           );
  C_5640_501_06_RYA601_SP_R0544 : FbAnalogValue_Medium (131) := (                _sDescription := 'Settpunkt',                 _rCov_Increment := 1,                 _eUnits := WagoTypesBacnet.eBACnetUnits.UNIT_PARTS_PER_MILLION           );
  C_5640_501_06_RYA601_MV_R0544 : FbAnalogInput_Large (43) := (                _sDescription := 'Målt CO2-konsentrasjon',                 _rCov_Increment := 1,                 _eUnits := WagoTypesBacnet.eBACnetUnits.UNIT_PARTS_PER_MILLION,                 _rHighLimit := 1000,                 _ILimitEnable := ( xLowLimitReporting := FALSE, xHighLimitReporting := TRUE ),                 _udiNotificationClass := 22           );
  C_5640_501_06_SBB01_C_R0544 : FbAnalogOutput_Medium (21) := (                _sDescription := 'Pådrag varmeorgan',                 _rCov_Increment := 1,                 _eUnits := WagoTypesBacnet.eBACnetUnits.UNIT_PERCENT           );
  C_5640_501_06_RMA6001_A1_R0401 : FbBinaryInput_Large (0) := (                _sDescription := 'Kommunikasjonsfeil'           );
  C_5640_501_06_RMA6002_A1_R0401 : FbBinaryInput_Large (1) := (                _sDescription := 'Kommunikasjonsfeil'           );
  C_5640_501_06_RMA6003_A1_R0406 : FbBinaryInput_Large (2) := (                _sDescription := 'Kommunikasjonsfeil'           );
  C_5640_501_06_RMA6004_A1_R0407 : FbBinaryInput_Large (3) := (                _sDescription := 'Kommunikasjonsfeil'           );
  C_5640_501_06_RMA6005_A1_R0408 : FbBinaryInput_Large (4) := (                _sDescription := 'Kommunikasjonsfeil'           );
  C_5640_501_06_RMA6006_A1_R0409 : FbBinaryInput_Large (5) := (                _sDescription := 'Kommunikasjonsfeil'           );
  C_5640_501_06_RMA6007_A1_R0409 : FbBinaryInput_Large (6) := (                _sDescription := 'Kommunikasjonsfeil'           );
  C_5640_501_06_RMA6008_A1_R0409 : FbBinaryInput_Large (7) := (                _sDescription := 'Kommunikasjonsfeil'           );
  C_5640_501_06_RMA6009_A1_R0464 : FbBinaryInput_Large (8) := (                _sDescription := 'Kommunikasjonsfeil'           );
  C_5640_501_06_RMA6010_A1_R0464 : FbBinaryInput_Large (9) := (                _sDescription := 'Kommunikasjonsfeil'           );
  C_5640_501_06_RMA6011_A1_R0415 : FbBinaryInput_Large (10) := (                _sDescription := 'Kommunikasjonsfeil'           );
  C_5640_501_06_RMA6012_A1_R0422 : FbBinaryInput_Large (11) := (                _sDescription := 'Kommunikasjonsfeil'           );
  C_5640_501_06_RMA6013_A1_R0422 : FbBinaryInput_Large (12) := (                _sDescription := 'Kommunikasjonsfeil'           );
  C_5640_501_06_RMA6014_A1_R0426_1 : FbBinaryInput_Large (13) := (                _sDescription := 'Kommunikasjonsfeil'           );
  C_5640_501_06_RMA6015_A1_R0426_2 : FbBinaryInput_Large (14) := (                _sDescription := 'Kommunikasjonsfeil'           );
  C_5640_501_06_RMA6016_A1_R0426_3 : FbBinaryInput_Large (15) := (                _sDescription := 'Kommunikasjonsfeil'           );
  C_5640_501_06_KAB6001_A1_R0401 : FbBinaryInput_Large (16) := (                _sDescription := 'Kommunikasjonsfeil'           );
  C_5640_501_06_KAB6002_A1_R0401 : FbBinaryInput_Large (17) := (                _sDescription := 'Kommunikasjonsfeil'           );
  C_5640_501_06_KAB6003_A1_R0401 : FbBinaryInput_Large (18) := (                _sDescription := 'Kommunikasjonsfeil'           );
  C_5640_501_06_KAB6004_A1_R0401 : FbBinaryInput_Large (19) := (                _sDescription := 'Kommunikasjonsfeil'           );
  C_5640_501_06_KAB6005_A1_R0401 : FbBinaryInput_Large (20) := (                _sDescription := 'Kommunikasjonsfeil'           );
  C_5640_501_06_KAB6006_A1_R0406 : FbBinaryInput_Large (21) := (                _sDescription := 'Kommunikasjonsfeil'           );
  C_5640_501_06_KAB6007_A1_R0406 : FbBinaryInput_Large (22) := (                _sDescription := 'Kommunikasjonsfeil'           );
  C_5640_501_06_KAB6008_A1_R0407 : FbBinaryInput_Large (23) := (                _sDescription := 'Kommunikasjonsfeil'           );
  C_5640_501_06_KAB6009_A1_R0407 : FbBinaryInput_Large (24) := (                _sDescription := 'Kommunikasjonsfeil'           );
  C_5640_501_06_KAB6010_A1_R0408 : FbBinaryInput_Large (25) := (                _sDescription := 'Kommunikasjonsfeil'           );
  C_5640_501_06_KAB6011_A1_R0409 : FbBinaryInput_Large (26) := (                _sDescription := 'Kommunikasjonsfeil'           );
  C_5640_501_06_KAB6012_A1_R0409 : FbBinaryInput_Large (27) := (                _sDescription := 'Kommunikasjonsfeil'           );
  C_5640_501_06_KAB6013_A1_R0409 : FbBinaryInput_Large (28) := (                _sDescription := 'Kommunikasjonsfeil'           );
  C_5640_501_06_KAB6014_A1_R0409 : FbBinaryInput_Large (29) := (                _sDescription := 'Kommunikasjonsfeil'           );
  C_5640_501_06_KAB6015_A1_R0409 : FbBinaryInput_Large (30) := (                _sDescription := 'Kommunikasjonsfeil'           );
  C_5640_501_06_KAB6016_A1_R0409 : FbBinaryInput_Large (31) := (                _sDescription := 'Kommunikasjonsfeil'           );
  C_5640_501_06_KAB6017_A1_R0409 : FbBinaryInput_Large (32) := (                _sDescription := 'Kommunikasjonsfeil'           );
  C_5640_501_06_KAB6018_A1_R0464 : FbBinaryInput_Large (33) := (                _sDescription := 'Kommunikasjonsfeil'           );
  C_5640_501_06_KAB6019_A1_R0464 : FbBinaryInput_Large (34) := (                _sDescription := 'Kommunikasjonsfeil'           );
  C_5640_501_06_KAB6020_A1_R0464 : FbBinaryInput_Large (35) := (                _sDescription := 'Kommunikasjonsfeil'           );
  C_5640_501_06_KAB6021_A1_R0464 : FbBinaryInput_Large (36) := (                _sDescription := 'Kommunikasjonsfeil'           );
  C_5640_501_06_KAB6022_A1_R0415 : FbBinaryInput_Large (37) := (                _sDescription := 'Kommunikasjonsfeil'           );
  C_5640_501_06_KAB6023_A1_R0415 : FbBinaryInput_Large (38) := (                _sDescription := 'Kommunikasjonsfeil'           );
  C_5640_501_06_KAB6024_A1_R0422 : FbBinaryInput_Large (39) := (                _sDescription := 'Kommunikasjonsfeil'           );
  C_5640_501_06_KAB6025_A1_R0422 : FbBinaryInput_Large (40) := (                _sDescription := 'Kommunikasjonsfeil'           );
  C_5640_501_06_KAB6026_A1_R0422 : FbBinaryInput_Large (41) := (                _sDescription := 'Kommunikasjonsfeil'           );
  C_5640_501_06_KAB6027_A1_R0422 : FbBinaryInput_Large (42) := (                _sDescription := 'Kommunikasjonsfeil'           );
  C_5640_501_06_KAB6028_A1_R0422 : FbBinaryInput_Large (43) := (                _sDescription := 'Kommunikasjonsfeil'           );
  C_5640_501_06_KAB6029_A1_R0426_1 : FbBinaryInput_Large (44) := (                _sDescription := 'Kommunikasjonsfeil'           );
  C_5640_501_06_KAB6030_A1_R0426_2 : FbBinaryInput_Large (45) := (                _sDescription := 'Kommunikasjonsfeil'           );
  C_5640_501_06_KAB6031_A1_R0426_3 : FbBinaryInput_Large (46) := (                _sDescription := 'Kommunikasjonsfeil'           );
  C_5640_501_06_RMA6001_A1_R0528 : FbBinaryInput_Large (47) := (                _sDescription := 'Kommunikasjonsfeil'           );
  C_5640_501_06_RMA6002_A1_R0523 : FbBinaryInput_Large (48) := (                _sDescription := 'Kommunikasjonsfeil'           );
  C_5640_501_06_RMA6003_A1_R0531 : FbBinaryInput_Large (49) := (                _sDescription := 'Kommunikasjonsfeil'           );
  C_5640_501_06_RMA6004_A1_R0535_1 : FbBinaryInput_Large (50) := (                _sDescription := 'Kommunikasjonsfeil'           );
  C_5640_501_06_RMA6005_A1_R0535_2 : FbBinaryInput_Large (51) := (                _sDescription := 'Kommunikasjonsfeil'           );
  C_5640_501_06_RMA6006_A1_R0535_3 : FbBinaryInput_Large (52) := (                _sDescription := 'Kommunikasjonsfeil'           );
  C_5640_501_06_RMA6007_A1_R0536 : FbBinaryInput_Large (53) := (                _sDescription := 'Kommunikasjonsfeil'           );
  C_5640_501_06_RMA6008_A1_R0543 : FbBinaryInput_Large (54) := (                _sDescription := 'Kommunikasjonsfeil'           );
  C_5640_501_06_RMA6009_A1_R0547_1 : FbBinaryInput_Large (55) := (                _sDescription := 'Kommunikasjonsfeil'           );
  C_5640_501_06_RMA6010_A1_R0547_2 : FbBinaryInput_Large (56) := (                _sDescription := 'Kommunikasjonsfeil'           );
  C_5640_501_06_RMA6011_A1_R0544 : FbBinaryInput_Large (57) := (                _sDescription := 'Kommunikasjonsfeil'           );
  C_5640_501_06_RMA6012_A1_R0544 : FbBinaryInput_Large (58) := (                _sDescription := 'Kommunikasjonsfeil'           );
  C_5640_501_06_KAB6001_A1_R0528 : FbBinaryInput_Large (59) := (                _sDescription := 'Kommunikasjonsfeil'           );
  C_5640_501_06_KAB6002_A1_R0523 : FbBinaryInput_Large (60) := (                _sDescription := 'Kommunikasjonsfeil'           );
  C_5640_501_06_KAB6003_A1_R0531 : FbBinaryInput_Large (61) := (                _sDescription := 'Kommunikasjonsfeil'           );
  C_5640_501_06_KAB6004_A1_R0531 : FbBinaryInput_Large (62) := (                _sDescription := 'Kommunikasjonsfeil'           );
  C_5640_501_06_KAB6005_A1_R0535_1 : FbBinaryInput_Large (63) := (                _sDescription := 'Kommunikasjonsfeil'           );
  C_5640_501_06_KAB6006_A1_R0535_1 : FbBinaryInput_Large (64) := (                _sDescription := 'Kommunikasjonsfeil'           );
  C_5640_501_06_KAB6007_A1_R0535_1 : FbBinaryInput_Large (65) := (                _sDescription := 'Kommunikasjonsfeil'           );
  C_5640_501_06_KAB6008_A1_R0535_1 : FbBinaryInput_Large (66) := (                _sDescription := 'Kommunikasjonsfeil'           );
  C_5640_501_06_KAB6009_A1_R0535_2 : FbBinaryInput_Large (67) := (                _sDescription := 'Kommunikasjonsfeil'           );
  C_5640_501_06_KAB6010_A1_R0535_2 : FbBinaryInput_Large (68) := (                _sDescription := 'Kommunikasjonsfeil'           );
  C_5640_501_06_KAB6011_A1_R0535_2 : FbBinaryInput_Large (69) := (                _sDescription := 'Kommunikasjonsfeil'           );
  C_5640_501_06_KAB6012_A1_R0535_2 : FbBinaryInput_Large (70) := (                _sDescription := 'Kommunikasjonsfeil'           );
  C_5640_501_06_KAB6013_A1_R0535_2 : FbBinaryInput_Large (71) := (                _sDescription := 'Kommunikasjonsfeil'           );
  C_5640_501_06_KAB6014_A1_R0535_2 : FbBinaryInput_Large (72) := (                _sDescription := 'Kommunikasjonsfeil'           );
  C_5640_501_06_KAB6015_A1_R0535_3 : FbBinaryInput_Large (73) := (                _sDescription := 'Kommunikasjonsfeil'           );
  C_5640_501_06_KAB6016_A1_R0535_3 : FbBinaryInput_Large (74) := (                _sDescription := 'Kommunikasjonsfeil'           );
  C_5640_501_06_KAB6017_A1_R0535_3 : FbBinaryInput_Large (75) := (                _sDescription := 'Kommunikasjonsfeil'           );
  C_5640_501_06_KAB6018_A1_R0536 : FbBinaryInput_Large (76) := (                _sDescription := 'Kommunikasjonsfeil'           );
  C_5640_501_06_KAB6019_A1_R0536 : FbBinaryInput_Large (77) := (                _sDescription := 'Kommunikasjonsfeil'           );
  C_5640_501_06_KAB6020_A1_R0543 : FbBinaryInput_Large (78) := (                _sDescription := 'Kommunikasjonsfeil'           );
  C_5640_501_06_KAB6021_A1_R0543 : FbBinaryInput_Large (79) := (                _sDescription := 'Kommunikasjonsfeil'           );
  C_5640_501_06_KAB6022_A1_R0547_1 : FbBinaryInput_Large (80) := (                _sDescription := 'Kommunikasjonsfeil'           );
  C_5640_501_06_KAB6023_A1_R0547_1 : FbBinaryInput_Large (81) := (                _sDescription := 'Kommunikasjonsfeil'           );
  C_5640_501_06_KAB6024_A1_R0547_1 : FbBinaryInput_Large (82) := (                _sDescription := 'Kommunikasjonsfeil'           );
  C_5640_501_06_KAB6025_A1_R0547_2 : FbBinaryInput_Large (83) := (                _sDescription := 'Kommunikasjonsfeil'           );
  C_5640_501_06_KAB6026_A1_R0547_2 : FbBinaryInput_Large (84) := (                _sDescription := 'Kommunikasjonsfeil'           );
  C_5640_501_06_KAB6027_A1_R0547_2 : FbBinaryInput_Large (85) := (                _sDescription := 'Kommunikasjonsfeil'           );
  C_5640_501_06_KAB6028_A1_R0544 : FbBinaryInput_Large (86) := (                _sDescription := 'Kommunikasjonsfeil'           );
  A_360_01_SQ4_A407_VOL : FbAnalogInput_Medium (2000) := (                _sDescription := 'Faktisk luftmengde',                 _rCov_Increment := 1,                 _eUnits := WagoTypesBacnet.eBACnetUnits.UNIT_CUBIC_METERS_PER_HOUR           );
  A_360_01_SQ4_A407_SP : FbAnalogValue_Medium (2000) := (                _sDescription := 'Settpunkt',                 _rCov_Increment := 1,                 _eUnits := WagoTypesBacnet.eBACnetUnits.UNIT_CUBIC_METERS_PER_HOUR           );
  A_360_01_SQ4_A407_VMIN : FbAnalogValue_Medium (2001) := (                _sDescription := 'Minste luftmengde',                 _rCov_Increment := 1,                 _eUnits := WagoTypesBacnet.eBACnetUnits.UNIT_CUBIC_METERS_PER_HOUR           );
  A_360_01_SQ4_A407_VMAX : FbAnalogValue_Medium (2002) := (                _sDescription := 'Største luftmengde',                 _rCov_Increment := 1,                 _eUnits := WagoTypesBacnet.eBACnetUnits.UNIT_CUBIC_METERS_PER_HOUR           );
  A_360_01_SQ4_A407_FB : FbAnalogInput_Medium (2001) := (                _sDescription := 'Spjeldvinkel',                 _rCov_Increment := 1,                 _eUnits := WagoTypesBacnet.eBACnetUnits.UNIT_PERCENT           );
  A_360_01_SQ4_A407_C : FbAnalogOutput_Medium (2000) := (                _sDescription := 'Pådrag',                 _rCov_Increment := 1,                 _eUnits := WagoTypesBacnet.eBACnetUnits.UNIT_PERCENT           );
  A_360_01_SQ4_A407_KMD : FbMultiStateValue_Large (2000) := (                _sDescription := 'Manuell overstyring',                 _udiNumberOfStates := 8           );
  A_360_01_SQ4_A407_OPT_EKSKL : FbBinaryValue_Medium (2000) := (                _sDescription := 'Optimizer',                 _sActiveText := 'Utkoblet',                 _sInactiveText := 'Innkoblet'           );
  A_360_01_SQ4_A407_A1 : FbBinaryInput_Large (2000) := (                _sDescription := 'Luftmengde Sjeld',                 _sActiveText := 'Feil på luftmengde',                 _sInactiveText := 'Ingen feil',                 _udiNotificationClass := 22           );
  A_360_01_SQ4_A407_A2 : FbBinaryInput_Large (2001) := (                _sDescription := 'Kommunikasjonovervåking',                 _sActiveText := 'Kommunikasjonsfeil',                 _sInactiveText := 'Ingen feil',                 _udiNotificationClass := 22           );
  A_360_01_SQ4_4AH2_VOL : FbAnalogInput_Medium (2002) := (                _sDescription := 'Faktisk luftmengde',                 _rCov_Increment := 1,                 _eUnits := WagoTypesBacnet.eBACnetUnits.UNIT_CUBIC_METERS_PER_HOUR           );
  A_360_01_SQ4_4AH2_SP : FbAnalogValue_Medium (2003) := (                _sDescription := 'Settpunkt',                 _rCov_Increment := 1,                 _eUnits := WagoTypesBacnet.eBACnetUnits.UNIT_CUBIC_METERS_PER_HOUR           );
  A_360_01_SQ4_4AH2_VMIN : FbAnalogValue_Medium (2004) := (                _sDescription := 'Minste luftmengde',                 _rCov_Increment := 1,                 _eUnits := WagoTypesBacnet.eBACnetUnits.UNIT_CUBIC_METERS_PER_HOUR           );
  A_360_01_SQ4_4AH2_VMAX : FbAnalogValue_Medium (2005) := (                _sDescription := 'Største luftmengde',                 _rCov_Increment := 1,                 _eUnits := WagoTypesBacnet.eBACnetUnits.UNIT_CUBIC_METERS_PER_HOUR           );
  A_360_01_SQ4_4AH2_FB : FbAnalogInput_Medium (2003) := (                _sDescription := 'Spjeldvinkel',                 _rCov_Increment := 1,                 _eUnits := WagoTypesBacnet.eBACnetUnits.UNIT_PERCENT           );
  A_360_01_SQ4_4AH2_C : FbAnalogOutput_Medium (2001) := (                _sDescription := 'Pådrag',                 _rCov_Increment := 1,                 _eUnits := WagoTypesBacnet.eBACnetUnits.UNIT_PERCENT           );
  A_360_01_SQ4_4AH2_KMD : FbMultiStateValue_Large (2001) := (                _sDescription := 'Manuell overstyring',                 _udiNumberOfStates := 8           );
  A_360_01_SQ4_4AH2_OPT_EKSKL : FbBinaryValue_Medium (2001) := (                _sDescription := 'Optimizer',                 _sActiveText := 'Utkoblet',                 _sInactiveText := 'Innkoblet'           );
  A_360_01_SQ4_4AH2_A1 : FbBinaryInput_Large (2002) := (                _sDescription := 'Luftmengde Sjeld',                 _sActiveText := 'Feil på luftmengde',                 _sInactiveText := 'Ingen feil',                 _udiNotificationClass := 22           );
  A_360_01_SQ4_4AH2_A2 : FbBinaryInput_Large (2003) := (                _sDescription := 'Kommunikasjonovervåking',                 _sActiveText := 'Kommunikasjonsfeil',                 _sInactiveText := 'Ingen feil',                 _udiNotificationClass := 22           );
  A_360_01_SQ4_4AH1_VOL : FbAnalogInput_Medium (2004) := (                _sDescription := 'Faktisk luftmengde',                 _rCov_Increment := 1,                 _eUnits := WagoTypesBacnet.eBACnetUnits.UNIT_CUBIC_METERS_PER_HOUR           );
  A_360_01_SQ4_4AH1_SP : FbAnalogValue_Medium (2006) := (                _sDescription := 'Settpunkt',                 _rCov_Increment := 1,                 _eUnits := WagoTypesBacnet.eBACnetUnits.UNIT_CUBIC_METERS_PER_HOUR           );
  A_360_01_SQ4_4AH1_VMIN : FbAnalogValue_Medium (2007) := (                _sDescription := 'Minste luftmengde',                 _rCov_Increment := 1,                 _eUnits := WagoTypesBacnet.eBACnetUnits.UNIT_CUBIC_METERS_PER_HOUR           );
  A_360_01_SQ4_4AH1_VMAX : FbAnalogValue_Medium (2008) := (                _sDescription := 'Største luftmengde',                 _rCov_Increment := 1,                 _eUnits := WagoTypesBacnet.eBACnetUnits.UNIT_CUBIC_METERS_PER_HOUR           );
  A_360_01_SQ4_4AH1_FB : FbAnalogInput_Medium (2005) := (                _sDescription := 'Spjeldvinkel',                 _rCov_Increment := 1,                 _eUnits := WagoTypesBacnet.eBACnetUnits.UNIT_PERCENT           );
  A_360_01_SQ4_4AH1_C : FbAnalogOutput_Medium (2002) := (                _sDescription := 'Pådrag',                 _rCov_Increment := 1,                 _eUnits := WagoTypesBacnet.eBACnetUnits.UNIT_PERCENT           );
  A_360_01_SQ4_4AH1_KMD : FbMultiStateValue_Large (2002) := (                _sDescription := 'Manuell overstyring',                 _udiNumberOfStates := 8           );
  A_360_01_SQ4_4AH1_OPT_EKSKL : FbBinaryValue_Medium (2002) := (                _sDescription := 'Optimizer',                 _sActiveText := 'Utkoblet',                 _sInactiveText := 'Innkoblet'           );
  A_360_01_SQ4_4AH1_A1 : FbBinaryInput_Large (2004) := (                _sDescription := 'Luftmengde Sjeld',                 _sActiveText := 'Feil på luftmengde',                 _sInactiveText := 'Ingen feil',                 _udiNotificationClass := 22           );
  A_360_01_SQ4_4AH1_A2 : FbBinaryInput_Large (2005) := (                _sDescription := 'Kommunikasjonovervåking',                 _sActiveText := 'Kommunikasjonsfeil',                 _sInactiveText := 'Ingen feil',                 _udiNotificationClass := 22           );
  A_360_01_SQ5_4AH1_VOL : FbAnalogInput_Medium (2006) := (                _sDescription := 'Faktisk luftmengde',                 _rCov_Increment := 1,                 _eUnits := WagoTypesBacnet.eBACnetUnits.UNIT_CUBIC_METERS_PER_HOUR           );
  A_360_01_SQ5_4AH1_SP : FbAnalogValue_Medium (2009) := (                _sDescription := 'Settpunkt',                 _rCov_Increment := 1,                 _eUnits := WagoTypesBacnet.eBACnetUnits.UNIT_CUBIC_METERS_PER_HOUR           );
  A_360_01_SQ5_4AH1_VMIN : FbAnalogValue_Medium (2010) := (                _sDescription := 'Minste luftmengde',                 _rCov_Increment := 1,                 _eUnits := WagoTypesBacnet.eBACnetUnits.UNIT_CUBIC_METERS_PER_HOUR           );
  A_360_01_SQ5_4AH1_VMAX : FbAnalogValue_Medium (2011) := (                _sDescription := 'Største luftmengde',                 _rCov_Increment := 1,                 _eUnits := WagoTypesBacnet.eBACnetUnits.UNIT_CUBIC_METERS_PER_HOUR           );
  A_360_01_SQ5_4AH1_FB : FbAnalogInput_Medium (2007) := (                _sDescription := 'Spjeldvinkel',                 _rCov_Increment := 1,                 _eUnits := WagoTypesBacnet.eBACnetUnits.UNIT_PERCENT           );
  A_360_01_SQ5_4AH1_C : FbAnalogOutput_Medium (2003) := (                _sDescription := 'Pådrag',                 _rCov_Increment := 1,                 _eUnits := WagoTypesBacnet.eBACnetUnits.UNIT_PERCENT           );
  A_360_01_SQ5_4AH1_KMD : FbMultiStateValue_Large (2003) := (                _sDescription := 'Manuell overstyring',                 _udiNumberOfStates := 8           );
  A_360_01_SQ5_4AH1_OPT_EKSKL : FbBinaryValue_Medium (2003) := (                _sDescription := 'Optimizer',                 _sActiveText := 'Utkoblet',                 _sInactiveText := 'Innkoblet'           );
  A_360_01_SQ5_4AH1_A1 : FbBinaryInput_Large (2006) := (                _sDescription := 'Luftmengde Sjeld',                 _sActiveText := 'Feil på luftmengde',                 _sInactiveText := 'Ingen feil',                 _udiNotificationClass := 22           );
  A_360_01_SQ5_4AH1_A2 : FbBinaryInput_Large (2007) := (                _sDescription := 'Kommunikasjonovervåking',                 _sActiveText := 'Kommunikasjonsfeil',                 _sInactiveText := 'Ingen feil',                 _udiNotificationClass := 22           );
  A_360_01_SQ5_A405_VOL : FbAnalogInput_Medium (2008) := (                _sDescription := 'Faktisk luftmengde',                 _rCov_Increment := 1,                 _eUnits := WagoTypesBacnet.eBACnetUnits.UNIT_CUBIC_METERS_PER_HOUR           );
  A_360_01_SQ5_A405_SP : FbAnalogValue_Medium (2012) := (                _sDescription := 'Settpunkt',                 _rCov_Increment := 1,                 _eUnits := WagoTypesBacnet.eBACnetUnits.UNIT_CUBIC_METERS_PER_HOUR           );
  A_360_01_SQ5_A405_VMIN : FbAnalogValue_Medium (2013) := (                _sDescription := 'Minste luftmengde',                 _rCov_Increment := 1,                 _eUnits := WagoTypesBacnet.eBACnetUnits.UNIT_CUBIC_METERS_PER_HOUR           );
  A_360_01_SQ5_A405_VMAX : FbAnalogValue_Medium (2014) := (                _sDescription := 'Største luftmengde',                 _rCov_Increment := 1,                 _eUnits := WagoTypesBacnet.eBACnetUnits.UNIT_CUBIC_METERS_PER_HOUR           );
  A_360_01_SQ5_A405_FB : FbAnalogInput_Medium (2009) := (                _sDescription := 'Spjeldvinkel',                 _rCov_Increment := 1,                 _eUnits := WagoTypesBacnet.eBACnetUnits.UNIT_PERCENT           );
  A_360_01_SQ5_A405_C : FbAnalogOutput_Medium (2004) := (                _sDescription := 'Pådrag',                 _rCov_Increment := 1,                 _eUnits := WagoTypesBacnet.eBACnetUnits.UNIT_PERCENT           );
  A_360_01_SQ5_A405_KMD : FbMultiStateValue_Large (2004) := (                _sDescription := 'Manuell overstyring',                 _udiNumberOfStates := 8           );
